// TwinCAT 3 PLC project SlaveController
// ProgramVersion: 3.1.4024.0
// libraries:
//   Tc2_EtherCAT, * (Beckhoff Automation GmbH)
//   Tc2_Math, * (Beckhoff Automation GmbH)
//   Tc2_Standard, * (Beckhoff Automation GmbH)
//   Tc2_System, * (Beckhoff Automation GmbH)
//   Tc2_Utilities, * (Beckhoff Automation GmbH)
//   Tc3_Module, * (Beckhoff Automation GmbH)
// project tree:
//   AgiMaths/Frames/ DHTrans.TcPOU, invFrame.TcPOU (not stored), rotX.TcPOU, rotY.TcPOU (not stored), rotZ.TcPOU (not stored), transform.TcPOU (not stored)
//   AgiMaths/MatrixLib/ angAxis2Rot.TcPOU, cross.TcPOU (not stored), Det5.TcPOU (not stored), Det6.TcPOU (not stored), Det7.TcPOU (not stored), invMat2.TcPOU, invMat6.TcPOU (not stored), invMat6Old.TcPOU (not stored), invMat3.TcPOU (not stored), invMat7.TcPOU, Mat3T.TcPOU (not stored), matAdd.TcPOU, matMultiNum.TcPOU (not stored), matMultiply.TcPOU (not stored), matMultiVec.TcPOU (not stored), matSelfAdd.TcPOU (not stored), vecDot.TcPOU (not stored), vecSelfAdd.TcPOU, matSelfSub.TcPOU (not stored), matSub.TcPOU (not stored), matTranspose.TcPOU (not stored), rot2AngAxis.TcPOU, vecAdd.TcPOU (not stored), norm.TcPOU, normalize.TcPOU, vecSelfMultiNum.TcPOU (not stored), vecMultiNum.TcPOU, vecSelfSub.TcPOU (not stored), vecSub.TcPOU (not stored)
//   AgiMaths/ sign.TcPOU (not stored), addVec7.TcPOU (not stored), atan2.TcPOU (not stored), cot.TcPOU (not stored)
//   DUTs/Enum/ E_ArmLightCtrlWord.TcDUT, E_CartJointState.TcDUT, E_EndoscopeType.TcDUT, E_EndoscopePosture.TcDUT, E_InstrumentType.TcDUT, E_MasterArmState.TcDUT, E_MatchedSlaveArmIdx.TcDUT (not stored), E_SetupArmState.TcDUT, E_SlaveArmState.TcDUT, E_DriverCtrlWord.TcDUT, E_DriverOPMode.TcDUT, E_DriverStatusWord.TcDUT
//   DUTs/Structure/MasterSlaveCommunication/ ST_MasterStatus.TcDUT, ST_SlaveStatus.TcDUT
//   DUTs/Structure/ ST_CartInputDataPool.TcDUT, ST_EtherCATState.TcDUT (not stored), ST_InstruOnChipData.TcDUT, ST_InstruStatus.TcDUT (not stored), ST_InstruTypeInfo.TcDUT, ST_SetupArmCtrlCmds.TcDUT (not stored), ST_SetupInputDataPool.TcDUT, ST_SlaveArmCtrlCmds.TcDUT, ST_SlaveInputDataPool.TcDUT, ST_Frame.TcDUT (not stored)
//   DUTs/Structure/TasksCommunication/ ST_CartJointData.TcDUT, ST_CartMotorInput.TcDUT, ST_CartMotorOutput.TcDUT, ST_CartStatus.TcDUT, ST_CartUIData.TcDUT, ST_SetupStatus.TcDUT, ST_SetupJointData.TcDUT, ST_SlaveDynaData.TcDUT, ST_SlaveUIData.TcDUT, ST_MasterJointData.TcDUT, ST_MotorInputs.TcDUT, ST_MotorOutputs.TcDUT, ST_SlaveJointData.TcDUT, ST_SafetyData.TcDUT
//   DUTs/Structure/UICommunication/ ST_cartOperation.TcDUT, ST_instruInfomation.TcDUT, ST_robotStateMachine.TcDUT, ST_uiControl.TcDUT
//   DUTs/Type/ Mat23.TcDUT, Mat2d.TcDUT, Mat32.TcDUT, Mat34.TcDUT (not stored), Mat53.TcDUT, Mat37.TcDUT (not stored), Mat43.TcDUT (not stored), Mat45.TcDUT (not stored), Mat35.TcDUT, Mat4d.TcDUT (not stored), Mat5d.TcDUT (not stored), Mat67.TcDUT (not stored), Mat6d.TcDUT (not stored), Mat76.TcDUT (not stored), Mat7d.TcDUT (not stored), Vec13d.TcDUT, Vec13di.TcDUT, Vec2d.TcDUT, Vec2i.TcDUT, Vec3i.TcDUT, Vec4b.TcDUT, Vec4d.TcDUT (not stored), Vec4i.TcDUT (not stored), Vec5b.TcDUT (not stored), Vec5d.TcDUT (not stored), Vec5i.TcDUT (not stored), Vec6b.TcDUT, Vec6i.TcDUT (not stored), Vec8b.TcDUT, Vec8d.TcDUT (not stored), Vec8di.TcDUT, Vec8i.TcDUT, Mat3d.TcDUT (not stored), Vec3d.TcDUT (not stored), Vec6d.TcDUT (not stored), Vec7d.TcDUT (not stored), Vec7i.TcDUT (not stored)
//   FBs_Auxiliary/ FB_cartJntDisenableDetect.TcPOU, FB_cartJntEnableDetect.TcPOU, FB_InstruNearDetect.TcPOU, FB_IOCheck.TcPOU, FB_IOToggleCheck.TcPOU, FB_rotaButtonDetect.TcPOU, FB_setupAdjustDetect.TcPOU, FB_setupJnt5AdjustDetect.TcPOU, FB_masterConnectionCheck.TcPOU, FB_TON.TcPOU (not stored), FB_trocarDetect.TcPOU, FB_PanelDetect.TcPOU (not stored), FB_InstrumentDetect.TcPOU, FB_AdjustDetect.TcPOU
//   FBs_BasicControllers/ FB_dither.TcPOU, FB_BasicInstruControl.TcPOU, FBMacroJntControl.TcPOU, FB_UltrosonicKnifeControl.TcPOU, FB_PID.TcPOU (not stored)
//   FBs_CartControlles/ FB_CartCtrlAdjust.TcPOU, FB_CartCtrlAsepticDeploy.TcPOU, FB_CartCtrlBase.TcPOU, FB_CartCtrlError.TcPOU, FB_CartCtrlInit.TcPOU, FB_CartCtrlInSurgery.TcPOU, FB_CartCtrlMotionCar.TcPOU, FB_CartCtrlReady.TcPOU, FB_CartCtrlRotaOverhang.TcPOU, FB_CartCtrlSlowDown.TcPOU, FB_CartCtrlStandColuAdjust.TcPOU, FB_CartPinDeploy.TcPOU, I_CartJointCtrl.TcIO
//   FBs_RobotDynamics/ FB_FullArmKinematic.TcPOU, FB_InstruViewCheck.TcPOU, FB_SlaveDynamic.TcPOU, FB_SlaveGravity.TcPOU, FB_SetupGravity.TcPOU
//   FBs_Robots/ FB_CartJoint.TcPOU, FB_CartRobot.TcPOU, FB_Instrument.TcPOU, FB_JointBase.TcPOU, FB_SetupArm.TcPOU, FB_SlaveCart.TcPOU, FB_SlaveJoint.TcPOU, FB_SetupJoint.TcPOU, FB_SetupRobot.TcPOU, FB_SlaveArm.TcPOU, FB_SlaveRobot.TcPOU
//   FBs_SetupControllers/ FB_SetupCtrlDisable.TcPOU, FB_SetupCtrlJnt5GraCali.TcPOU, FB_SetupCtrlHold.TcPOU, FB_SetupCtrlManualAdjust.TcPOU, FB_SetupCtrlPerformance.TcPOU, FB_SetupArmCtrlBase.TcPOU, FB_SetupCtrlAutoAdjust.TcPOU, FB_SetupCtrlCart.TcPOU (not stored), FB_SetupCtrlError.TcPOU, FB_SetupCtrlJnt3GraCali.TcPOU, FB_SetupCtrlInit.TcPOU, FB_SetupCtrlPackage.TcPOU (not stored), FB_SetupCtrlSelfCheck.TcPOU, I_SetupArmCtrl.TcIO (not stored)
//   FBs_SlaveControllers/ FB_SlaveCtrlDisable.TcPOU, FB_SlaveCtrlInstruInvasion.TcPOU, FB_SlaveCtrlInstruRetract.TcPOU, FB_SlaveCtrlInstruCali.TcPOU, FB_SlaveCtrlPerformance.TcPOU, FB_SlaveCtrlScopeToggle.TcPOU, FB_SlaveCtrlStop.TcPOU, FB_SlaveCtrlTest.TcPOU, FB_SlaveCtrlPackage.TcPOU, FB_SlaveCtrlEndoscope.TcPOU, FB_SlaveCtrlCart.TcPOU, FB_SlaveCtrlScopeReady.TcPOU, FB_SlaveCtrlSelfCheck.TcPOU, FB_SlaveCtrlError.TcPOU, FB_SlaveCtrlInstruReady.TcPOU, FB_SlaveCtrlMasterSlave.TcPOU, FB_SlaveCtrlMountInstru.TcPOU, FB_SlaveCtrlAdjust.TcPOU, FB_SlaveCtrlMountPanel.TcPOU, FB_SlaveCtrlPanelReady.TcPOU, FB_SlaveCtrlGraCali.TcPOU, FB_SlaveCtrlInit.TcPOU, FB_SlaveCtrlStandBy.TcPOU, FB_SlaveArmCtrlBase.TcPOU, I_SlaveArmCtrl.TcIO
//   FBs_TrajectoryPlanning/ FB_BasicDoubleS.TcPOU (not stored), FB_trajBase.TcPOU (not stored), FB_TrajMoveJ.TcPOU, FB_setupTrajMoveJ.TcPOU, linear_trajectory_with_quintic_polynomial_blends.TcPOU (not stored), quintic_spline_curve.TcPOU (not stored), Quintic_spline_curve_factor.TcPOU (not stored), TrapezoIDal_velocity_trajectory.TcPOU (not stored)
//   FBs_TrajectoryPlanning/OTG/ FB_secOrdTrajFilter.TcPOU (not stored), FB_thirdOrdTrajFilter.TcPOU (not stored)
//   FBs_Filters/ FB_LowPassFilter.TcPOU (not stored)
//   GVLs/CartJoints/ GVL_CartControlParameters.TcGVL, GVL_CartJointEncoderCaliData.TcGVL, GVL_CartMotorParameters.TcGVL
//   GVLs/configs/robot3/ GVL_CartJointEncoderCaliData_3.TcGVL, GVL_SetupArmDynamics_3.TcGVL, GVL_SlaveArmDynamics_3.TcGVL, GVL_SetupJointEncoderCaliData_3.TcGVL, GVL_SlaveJointEncoderCaliData_3.TcGVL
//   GVLs/configs/robot5/ GVL_CartJointEncoderCaliData_5.TcGVL, GVL_SetupArmDynamics_5.TcGVL, GVL_SlaveArmDynamics_5.TcGVL, GVL_SetupJointEncoderCaliData_5.TcGVL, GVL_SlaveJointEncoderCaliData_5.TcGVL
//   GVLs/configs/robot4/ GVL_SetupArmDynamics_4.TcGVL, GVL_SetupJointEncoderCaliData_4.TcGVL (not stored), GVL_SlaveArmDynamics_4.TcGVL, GVL_SlaveJointEncoderCaliData_4.TcGVL
//   GVLs/configs/robot6/ GVL_CartJointEncoderCaliData_6.TcGVL, GVL_SetupArmDynamics_6.TcGVL, GVL_SetupJointEncoderCaliData_6.TcGVL, GVL_SlaveArmDynamics_6.TcGVL, GVL_SlaveJointEncoderCaliData_6.TcGVL
//   GVLs/ GVL_interactUI.TcGVL, GVL_MathDefine.TcGVL, GVL_SafetyLogData.TcGVL, GVL_SafetyParameters.TcGVL, GVL_SystemParameters.TcGVL
//   GVLs/Instrument/ GVL_InstruCtrlParams.TcGVL, GVL_InstruTypeDefine.TcGVL
//   GVLs/SetupArms/ GVL_SetupArmDynamics.TcGVL, GVL_SetupJointEncoderCaliData.TcGVL, GVL_SetupMotorParameters.TcGVL, GVL_SetupArmKinematic.TcGVL, GVL_SetupControlParameters.TcGVL
//   GVLs/SlaveArms/ GVL_SlaveArmDynamics.TcGVL, GVL_SlaveArmKinematic.TcGVL, GVL_SlaveControlParameters.TcGVL, GVL_SlaveJointEncoderCaliData.TcGVL, GVL_SlaveMotorParameters.TcGVL
//   Mains/ CartControl.TcPOU, SafetyCheck.TcPOU, SetupArmControl.TcPOU (not stored), SlaveArmControl.TcPOU, RobotDynamics.TcPOU
//   SafetyCheck/ ASSERT.TcPOU, Fb_dataRecord.TcPOU, FB_EtherCATCheck.TcPOU (not stored), Fb_SafetyCheck.TcPOU, FB_Writer.TcPOU (not stored)
//   SafetyCheck/ErrRecord/ checkDelay.TcDUT, checkDelayTime.TcDUT, checkInputVariable.TcDUT, checkPermit.TcDUT, ST_Buffer.TcDUT, T_Buffer.TcDUT
//   Sandbox/ FB_SetupArmCheck.TcPOU (not stored), FB_SlaveArmCheck.TcPOU, FB_SlaveCtrlAdjust_bak1.TcPOU, FB_SlaveCtrlMasterSlave_bak1.TcPOU, FB_SlaveCtrlMasterSlave_bak2.TcPOU
//   Sandbox/knifeCmdPoseTest/ atan2_function.TcPOU, FB_CSVWrite.TcPOU, knifePoseSelect.TcPOU, tr_to_rpy.TcPOU, tr_to_space_vector.TcPOU
//   / TaskCartControl.TcTTO, TaskDynamic.TcTTO (not stored), TaskSafetyCheck.TcTTO, TaskSetupArmControl.TcTTO (not stored), TaskSlaveArmControl.TcTTO
// real-time tasks:
//   TASK TaskSlaveArmControl: cycle T#250us, priority 1, ADS port 350
//   TASK TaskDynamic: cycle T#1ms, priority 2, ADS port 351
//   TASK TaskSetupArmControl: cycle T#1ms, priority 3, ADS port 352
//   TASK TaskSafetyCheck: cycle T#1ms, priority 6, ADS port 353
//   TASK TaskCartControl: cycle T#1ms, priority 4, ADS port 354
// I/O:
//   DEVICE Device 5 (RT-Ethernet Adapter)
//   DEVICE MSCommunication, AmsNetId 169.254.186.39.2.1
//     Term 20 (EK1100) [EK1100 EtherCAT Coupler (2A E-Bus)]
//       Term 21 (EL6695) [EL6695 EtherCAT Bridge terminal (Primary)]
//       Term 8 (EL9011) [EL9011 End Terminal]
//     Term 22 (EK1100) [EK1100 EtherCAT Coupler (2A E-Bus)]
//       Term 23 (EL6070) [EL6070 1Ch. Licensing-Terminal]
//       Term 24 (EL1008) [EL1008 8Ch. Dig. Input 24V, 3ms]
//       Term 25 (EL2008) [EL2008 8Ch. Dig. Output 24V, 0.5A]
//       Term 26 (EL3004) [EL3004 4Ch. Ana. Input +/-10V]
//       Term 9 (EL9011) [EL9011 End Terminal]
//   DEVICE SlaveArm1, AmsNetId 169.254.186.39.3.1
//     Box 29 (CU2508) [CU2508 Ethernet Port]
//     SetupJoint12 [AX58200_MotorControl]
//     SetupJoint3 [AX58200_MotorControl]
//     SetupJoint4 [AX58200_MotorControl]
//     SetupJoint5 [AX58200_MotorControl]
//     SlaveJoint1 [AX58200_MotorControl]
//     SlaveJoint2 [AX58200_MotorControl]
//     SlaveJoint3 [AX58200_MotorControl]
//     SlaveJoint45 [AX58200_MotorControl]
//     SlaveJoint678 [AX58200_MotorControl]
//   DEVICE SlaveArm2, AmsNetId 169.254.186.39.8.1
//     Box 39 (CU2508) [CU2508 Ethernet Port]
//     SetupJoint12 [AX58200_MotorControl]
//     SetupJoint3 [AX58200_MotorControl]
//     SetupJoint4 [AX58200_MotorControl]
//     SetupJoint5 [AX58200_MotorControl]
//     SlaveJoint1 [AX58200_MotorControl]
//     SlaveJoint2 [AX58200_MotorControl]
//     SlaveJoint3 [AX58200_MotorControl]
//     SlaveJoint45 [AX58200_MotorControl]
//     SlaveJoint678 [AX58200_MotorControl]
//   DEVICE SlaveArm3, AmsNetId 169.254.186.39.9.1
//     Box 49 (CU2508) [CU2508 Ethernet Port]
//     SetupJoint12 [AX58200_MotorControl]
//     SetupJoint3 [AX58200_MotorControl]
//     SetupJoint4 [AX58200_MotorControl]
//     SetupJoint5 [AX58200_MotorControl]
//     SlaveJoint1 [AX58200_MotorControl]
//     SlaveJoint2 [AX58200_MotorControl]
//     SlaveJoint3 [AX58200_MotorControl]
//     SlaveJoint45 [AX58200_MotorControl]
//     SlaveJoint678 [AX58200_MotorControl]
//   DEVICE SlaveArm4, AmsNetId 169.254.186.39.10.1
//     Box 59 (CU2508) [CU2508 Ethernet Port]
//     SetupJoint12 [AX58200_MotorControl]
//     SetupJoint3 [AX58200_MotorControl]
//     SetupJoint4 [AX58200_MotorControl]
//     SetupJoint5 [AX58200_MotorControl]
//     SlaveJoint1 [AX58200_MotorControl]
//     SlaveJoint2 [AX58200_MotorControl]
//     SlaveJoint3 [AX58200_MotorControl_3AxiS]
//     SlaveJoint45 [AX58200_MotorControl_3AxiS]
//     SlaveJoint678 [AX58200_MotorControl_3AxiS]
//   DEVICE Cart, AmsNetId 169.254.186.39.4.1
//     CartJnt5 [iPOS8015 BZ-CAT]
//     CartJnt3 [iPOS4850 BX-CAT]
//     CartJnt4 [iPOS4850 BX-CAT]
//     CartJnt1 [AX58200_MotorControl]
//     CartJnt2 [AX58200_MotorControl]
//     CartJnt6 [AX58200_MotorControl]
//     CartJnt7 [AX58200_MotorControl]
//     CartJnt8 [AX58200_MotorControl]
// variable links:
//   SlaveController/SlaveController Instance <-> Cart/CartJnt1
//     TaskCartControl Inputs/CartControl.m_cartRobot.m_slaveCart.m_cartJoints[1].m_motorInputs/m_current <-> TxPdoMappingCspCsv/Torque actual value
//     TaskCartControl Inputs/CartControl.m_cartRobot.m_slaveCart.m_cartJoints[1].m_motorInputs/m_driverError <-> TxPdoMappingCspCsv/digital input
//     TaskCartControl Inputs/CartControl.m_cartRobot.m_slaveCart.m_cartJoints[1].m_motorInputs/m_motorEncoder <-> TxPdoMappingCspCsv/Position actual value
//     TaskCartControl Inputs/CartControl.m_cartRobot.m_slaveCart.m_cartJoints[1].m_motorInputs/m_statusWord <-> TxPdoMappingCspCsv/Statusword
//     TaskCartControl Outputs/CartControl.m_cartRobot.m_slaveCart.m_cartJoints[1].m_motorOutputs/m_cmdCurrent <-> RxPdoMappingCspCsv/Target torque
//     TaskCartControl Outputs/CartControl.m_cartRobot.m_slaveCart.m_cartJoints[1].m_motorOutputs/m_cmdMotorEncoder <-> RxPdoMappingCspCsv/Target position
//     TaskCartControl Outputs/CartControl.m_cartRobot.m_slaveCart.m_cartJoints[1].m_motorOutputs/m_controlWord <-> RxPdoMappingCspCsv/Controlword
//     TaskCartControl Outputs/CartControl.m_cartRobot.m_slaveCart.m_cartJoints[1].m_motorOutputs/m_opMode <-> RxPdoMappingCspCsv/Modes of operation
//   SlaveController/SlaveController Instance <-> Cart/CartJnt2
//     TaskCartControl Inputs/CartControl.m_cartRobot.m_slaveCart.m_cartJoints[2].m_motorInputs/m_current <-> TxPdoMappingCspCsv/Torque actual value
//     TaskCartControl Inputs/CartControl.m_cartRobot.m_slaveCart.m_cartJoints[2].m_motorInputs/m_driverError <-> TxPdoMappingCspCsv/digital input
//     TaskCartControl Inputs/CartControl.m_cartRobot.m_slaveCart.m_cartJoints[2].m_motorInputs/m_motorEncoder <-> TxPdoMappingCspCsv/Position actual value
//     TaskCartControl Inputs/CartControl.m_cartRobot.m_slaveCart.m_cartJoints[2].m_motorInputs/m_statusWord <-> TxPdoMappingCspCsv/Statusword
//     TaskCartControl Inputs/CartControl.m_cartRobot.m_slaveCart.m_cartJoints[5].m_motorInputs/m_linkEncoder <-> TxPdoMappingCspCsv/ENC2
//     TaskCartControl Outputs/CartControl.m_cartRobot.m_slaveCart.m_cartJoints[2].m_motorOutputs/m_cmdCurrent <-> RxPdoMappingCspCsv/Target torque
//     TaskCartControl Outputs/CartControl.m_cartRobot.m_slaveCart.m_cartJoints[2].m_motorOutputs/m_cmdMotorEncoder <-> RxPdoMappingCspCsv/Target position
//     TaskCartControl Outputs/CartControl.m_cartRobot.m_slaveCart.m_cartJoints[2].m_motorOutputs/m_controlWord <-> RxPdoMappingCspCsv/Controlword
//     TaskCartControl Outputs/CartControl.m_cartRobot.m_slaveCart.m_cartJoints[2].m_motorOutputs/m_opMode <-> RxPdoMappingCspCsv/Modes of operation
//   SlaveController/SlaveController Instance <-> Cart/CartJnt3
//     TaskCartControl Inputs/CartControl.m_cartRobot.m_slaveCart.m_cartJoints[3].m_motorInputs/m_motorEncoder <-> Transmit PDO 1 mapping parameters/Position actual value
//     TaskCartControl Inputs/CartControl.m_cartRobot.m_slaveCart.m_cartJoints[3].m_motorInputs/m_statusWord <-> Transmit PDO 1 mapping parameters/Statusword
//     TaskCartControl Outputs/CartControl.m_cartRobot.m_slaveCart.m_cartJoints[3].m_cartMotorOutput/m_cmdAccMz <-> Receive PDO 4 mapping parameters/Profile acceleration
//     TaskCartControl Outputs/CartControl.m_cartRobot.m_slaveCart.m_cartJoints[3].m_cartMotorOutput/m_cmdVelMz <-> Receive PDO 4 mapping parameters/Profile velocity
//     TaskCartControl Outputs/CartControl.m_cartRobot.m_slaveCart.m_cartJoints[3].m_cartMotorOutput/m_cmdVelMzVelMode <-> Receive PDO 3 mapping parameters/Target Velocity
//     TaskCartControl Outputs/CartControl.m_cartRobot.m_slaveCart.m_cartJoints[3].m_motorOutputs/m_cmdMotorEncoder <-> Receive PDO 1 mapping parameters/Target position
//     TaskCartControl Outputs/CartControl.m_cartRobot.m_slaveCart.m_cartJoints[3].m_motorOutputs/m_controlWord <-> Receive PDO 1 mapping parameters/Controlword
//     TaskCartControl Outputs/CartControl.m_cartRobot.m_slaveCart.m_cartJoints[3].m_motorOutputs/m_opMode <-> Receive PDO 3 mapping parameters/Modes of operation
//   SlaveController/SlaveController Instance <-> Cart/CartJnt4
//     TaskCartControl Inputs/CartControl.m_cartRobot.m_slaveCart.m_cartJoints[4].m_motorInputs/m_motorEncoder <-> Transmit PDO 1 mapping parameters/Position actual value
//     TaskCartControl Inputs/CartControl.m_cartRobot.m_slaveCart.m_cartJoints[4].m_motorInputs/m_statusWord <-> Transmit PDO 1 mapping parameters/Statusword
//     TaskCartControl Outputs/CartControl.m_cartRobot.m_slaveCart.m_cartJoints[4].m_cartMotorOutput/m_cmdAccMz <-> Receive PDO 4 mapping parameters/Profile acceleration
//     TaskCartControl Outputs/CartControl.m_cartRobot.m_slaveCart.m_cartJoints[4].m_cartMotorOutput/m_cmdVelMz <-> Receive PDO 4 mapping parameters/Profile velocity
//     TaskCartControl Outputs/CartControl.m_cartRobot.m_slaveCart.m_cartJoints[4].m_cartMotorOutput/m_cmdVelMzVelMode <-> Receive PDO 3 mapping parameters/Target  Velocity
//     TaskCartControl Outputs/CartControl.m_cartRobot.m_slaveCart.m_cartJoints[4].m_motorOutputs/m_cmdMotorEncoder <-> Receive PDO 1 mapping parameters/Target position
//     TaskCartControl Outputs/CartControl.m_cartRobot.m_slaveCart.m_cartJoints[4].m_motorOutputs/m_controlWord <-> Receive PDO 1 mapping parameters/Controlword
//     TaskCartControl Outputs/CartControl.m_cartRobot.m_slaveCart.m_cartJoints[4].m_motorOutputs/m_opMode <-> Receive PDO 3 mapping parameters/Modes of operation
//   SlaveController/SlaveController Instance <-> Cart/CartJnt5
//     TaskCartControl Inputs/CartControl.m_cartRobot.m_slaveCart.m_cartJoints[5].m_motorInputs/m_motorEncoder <-> Transmit PDO 1 mapping parameters/Position actual value
//     TaskCartControl Inputs/CartControl.m_cartRobot.m_slaveCart.m_cartJoints[5].m_motorInputs/m_statusWord <-> Transmit PDO 1 mapping parameters/Statusword
//     TaskCartControl Outputs/CartControl.m_cartRobot.m_slaveCart.m_cartJoints[5].m_cartMotorOutput/m_cmdAccMz <-> Receive PDO 4 mapping parameters/Profile acceleration
//     TaskCartControl Outputs/CartControl.m_cartRobot.m_slaveCart.m_cartJoints[5].m_cartMotorOutput/m_cmdVelMz <-> Receive PDO 4 mapping parameters/Profile velocity
//     TaskCartControl Outputs/CartControl.m_cartRobot.m_slaveCart.m_cartJoints[5].m_cartMotorOutput/m_cmdVelMzVelMode <-> Receive PDO 3 mapping parameters/Target Velocity
//     TaskCartControl Outputs/CartControl.m_cartRobot.m_slaveCart.m_cartJoints[5].m_motorOutputs/m_cmdMotorEncoder <-> Receive PDO 1 mapping parameters/Target position
//     TaskCartControl Outputs/CartControl.m_cartRobot.m_slaveCart.m_cartJoints[5].m_motorOutputs/m_controlWord <-> Receive PDO 1 mapping parameters/Controlword
//     TaskCartControl Outputs/CartControl.m_cartRobot.m_slaveCart.m_cartJoints[5].m_motorOutputs/m_opMode <-> Receive PDO 3 mapping parameters/Modes of operation
//   SlaveController/SlaveController Instance <-> Cart/CartJnt6
//     TaskCartControl Inputs/CartControl.m_cartRobot.m_slaveCart.m_cartJoints[6].m_motorInputs/m_current <-> TxPdoMappingCspCsv/Torque actual value
//     TaskCartControl Inputs/CartControl.m_cartRobot.m_slaveCart.m_cartJoints[6].m_motorInputs/m_driverError <-> TxPdoMappingCspCsv/digital input
//     TaskCartControl Inputs/CartControl.m_cartRobot.m_slaveCart.m_cartJoints[6].m_motorInputs/m_linkEncoder <-> TxPdoMappingCspCsv/ENC2
//     TaskCartControl Inputs/CartControl.m_cartRobot.m_slaveCart.m_cartJoints[6].m_motorInputs/m_motorEncoder <-> TxPdoMappingCspCsv/Position actual value
//     TaskCartControl Inputs/CartControl.m_cartRobot.m_slaveCart.m_cartJoints[6].m_motorInputs/m_statusWord <-> TxPdoMappingCspCsv/Statusword
//     TaskCartControl Outputs/CartControl.m_cartRobot.m_openHorizonLaser <-> RxPdoMappingCspCsv/Target velocity
//     TaskCartControl Outputs/CartControl.m_cartRobot.m_slaveCart.m_cartJoints[6].m_motorOutputs/m_cmdCurrent <-> RxPdoMappingCspCsv/Target torque
//     TaskCartControl Outputs/CartControl.m_cartRobot.m_slaveCart.m_cartJoints[6].m_motorOutputs/m_cmdMotorEncoder <-> RxPdoMappingCspCsv/Target position
//     TaskCartControl Outputs/CartControl.m_cartRobot.m_slaveCart.m_cartJoints[6].m_motorOutputs/m_controlWord <-> RxPdoMappingCspCsv/Controlword
//     TaskCartControl Outputs/CartControl.m_cartRobot.m_slaveCart.m_cartJoints[6].m_motorOutputs/m_opMode <-> RxPdoMappingCspCsv/Modes of operation
//   SlaveController/SlaveController Instance <-> Cart/CartJnt7
//     TaskCartControl Inputs/CartControl.m_cartRobot.m_slaveCart.m_cartJoints[7].m_motorInputs/m_current <-> TxPdoMappingCspCsv/Torque actual value
//     TaskCartControl Inputs/CartControl.m_cartRobot.m_slaveCart.m_cartJoints[7].m_motorInputs/m_driverError <-> TxPdoMappingCspCsv/digital input
//     TaskCartControl Inputs/CartControl.m_cartRobot.m_slaveCart.m_cartJoints[7].m_motorInputs/m_linkEncoder <-> TxPdoMappingCspCsv/ENC2
//     TaskCartControl Inputs/CartControl.m_cartRobot.m_slaveCart.m_cartJoints[7].m_motorInputs/m_motorEncoder <-> TxPdoMappingCspCsv/Position actual value
//     TaskCartControl Inputs/CartControl.m_cartRobot.m_slaveCart.m_cartJoints[7].m_motorInputs/m_statusWord <-> TxPdoMappingCspCsv/Statusword
//     TaskCartControl Outputs/CartControl.m_cartRobot.m_slaveCart.m_cartJoints[7].m_motorOutputs/m_cmdCurrent <-> RxPdoMappingCspCsv/Target torque
//     TaskCartControl Outputs/CartControl.m_cartRobot.m_slaveCart.m_cartJoints[7].m_motorOutputs/m_cmdMotorEncoder <-> RxPdoMappingCspCsv/Target position
//     TaskCartControl Outputs/CartControl.m_cartRobot.m_slaveCart.m_cartJoints[7].m_motorOutputs/m_controlWord <-> RxPdoMappingCspCsv/Controlword
//     TaskCartControl Outputs/CartControl.m_cartRobot.m_slaveCart.m_cartJoints[7].m_motorOutputs/m_opMode <-> RxPdoMappingCspCsv/Modes of operation
//   SlaveController/SlaveController Instance <-> Cart/CartJnt8
//     TaskCartControl Inputs/CartControl.m_cartRobot.m_slaveCart.m_cartJoints[8].m_motorInputs/m_current <-> TxPdoMappingCspCsv/Torque actual value
//     TaskCartControl Inputs/CartControl.m_cartRobot.m_slaveCart.m_cartJoints[8].m_motorInputs/m_driverError <-> TxPdoMappingCspCsv/digital input
//     TaskCartControl Inputs/CartControl.m_cartRobot.m_slaveCart.m_cartJoints[8].m_motorInputs/m_linkEncoder <-> TxPdoMappingCspCsv/ENC2
//     TaskCartControl Inputs/CartControl.m_cartRobot.m_slaveCart.m_cartJoints[8].m_motorInputs/m_motorEncoder <-> TxPdoMappingCspCsv/Position actual value
//     TaskCartControl Inputs/CartControl.m_cartRobot.m_slaveCart.m_cartJoints[8].m_motorInputs/m_statusWord <-> TxPdoMappingCspCsv/Statusword
//     TaskCartControl Outputs/CartControl.m_cartRobot.m_openCrossLaser <-> RxPdoMappingCspCsv/Target velocity
//     TaskCartControl Outputs/CartControl.m_cartRobot.m_slaveCart.m_cartJoints[8].m_motorOutputs/m_cmdCurrent <-> RxPdoMappingCspCsv/Target torque
//     TaskCartControl Outputs/CartControl.m_cartRobot.m_slaveCart.m_cartJoints[8].m_motorOutputs/m_cmdMotorEncoder <-> RxPdoMappingCspCsv/Target position
//     TaskCartControl Outputs/CartControl.m_cartRobot.m_slaveCart.m_cartJoints[8].m_motorOutputs/m_controlWord <-> RxPdoMappingCspCsv/Controlword
//     TaskCartControl Outputs/CartControl.m_cartRobot.m_slaveCart.m_cartJoints[8].m_motorOutputs/m_opMode <-> RxPdoMappingCspCsv/Modes of operation
//   SlaveController/SlaveController Instance <-> MSCommunication/Term 20 (EK1100)/Term 21 (EL6695)
//     TaskSafetyCheck Inputs/SafetyCheck.m_masterRobotData <-> IO Inputs/MasterRobotData
//     TaskSlaveArmControl Inputs/SlaveArmControl.m_masterRobotData <-> IO Inputs/MasterRobotData
//     TaskSlaveArmControl Outputs/SlaveArmControl.m_slaveRobotData <-> IO Outputs/SlaveRobotData
//   SlaveController/SlaveController Instance <-> MSCommunication/Term 22 (EK1100)/Term 24 (EL1008)
//     TaskCartControl Inputs/CartControl.m_cartRobot.m_carHandChassisDriveUnlock[1] <-> Channel 5/Input
//     TaskCartControl Inputs/CartControl.m_cartRobot.m_carHandChassisDriveUnlock[2] <-> Channel 6/Input
//     TaskCartControl Inputs/CartControl.m_cartRobot.m_slaveCart.m_drivingLeverSensorAuto <-> Channel 8/Input
//     TaskCartControl Inputs/CartControl.m_cartRobot.m_slaveCart.m_drivingLeverSensorManual <-> Channel 7/Input
//     TaskCartControl Inputs/CartControl.m_cartRobot.m_slaveCart.m_stabilizFootSensorLeft <-> Channel 3/Input
//     TaskCartControl Inputs/CartControl.m_cartRobot.m_slaveCart.m_stabilizFootSensorRight <-> Channel 4/Input
//     TaskSafetyCheck Inputs/SafetyCheck.m_emergencyStopButton <-> Channel 2/Input
//     TaskSlaveArmControl Inputs/SafetyCheck.m_stopButton <-> Channel 1/Input
//   SlaveController/SlaveController Instance <-> MSCommunication/Term 22 (EK1100)/Term 25 (EL2008)
//     TaskCartControl Outputs/CartControl.m_cartRobot.m_slaveCart.m_screwBreak <-> Channel 5/Output
//     TaskSafetyCheck Outputs/SafetyCheck.m_warningTone[{1..4}] <-> Channel {1..4}/Output  (4 links)
//   SlaveController/SlaveController Instance <-> MSCommunication/Term 22 (EK1100)/Term 26 (EL3004)
//     TaskCartControl Inputs/CartControl.m_cartRobot.m_slaveCart.m_driveForce[1] <-> AI Standard Channel 2/Value
//     TaskCartControl Inputs/CartControl.m_cartRobot.m_slaveCart.m_driveForce[2] <-> AI Standard Channel 1/Value
//   SlaveController/SlaveController Instance <-> SlaveArm1/SetupJoint12
//     TaskSetupArmControl Inputs/SetupArmControl.m_setupRobot.m_setupArms[1].m_joints[1].m_motorInputs/m_linkEncoder <-> TxPdoMappingCspCsv/ENC2
//     TaskSetupArmControl Inputs/SetupArmControl.m_setupRobot.m_setupArms[1].m_joints[1].m_motorInputs/m_statusWord <-> TxPdoMappingCspCsv/Statusword
//     TaskSetupArmControl Inputs/SetupArmControl.m_setupRobot.m_setupArms[1].m_joints[2].m_motorInputs/m_statusWord <-> TxPdoMappingCspCsv/Statusword
//     TaskSetupArmControl Inputs/SetupArmControl.m_setupRobot.m_setupArms[1].m_joints[2].m_motorInputs/m_linkEncoder <-> TxPdoMappingCspCsv/Torque actual value
//     TaskSetupArmControl Outputs/SetupArmControl.m_setupRobot.m_setupArms[1].m_joints[1].m_motorOutputs/m_controlWord <-> RxPdoMappingCspCsv/Controlword
//   SlaveController/SlaveController Instance <-> SlaveArm1/SetupJoint3
//     TaskSetupArmControl Inputs/SetupArmControl.m_setupRobot.m_setupArms[1].m_joints[3].m_motorInputs/m_current <-> TxPdoMappingCspCsv/Torque actual value
//     TaskSetupArmControl Inputs/SetupArmControl.m_setupRobot.m_setupArms[1].m_joints[3].m_motorInputs/m_linkEncoder <-> TxPdoMappingCspCsv/ENC2
//     TaskSetupArmControl Inputs/SetupArmControl.m_setupRobot.m_setupArms[1].m_joints[3].m_motorInputs/m_motorEncoder <-> TxPdoMappingCspCsv/Position actual value
//     TaskSetupArmControl Inputs/SetupArmControl.m_setupRobot.m_setupArms[1].m_joints[3].m_motorInputs/m_statusWord <-> TxPdoMappingCspCsv/Statusword
//     TaskSetupArmControl Outputs/SetupArmControl.m_setupRobot.m_setupArms[1].m_joints[3].m_motorOutputs/m_cmdCurrent <-> RxPdoMappingCspCsv/Target torque
//     TaskSetupArmControl Outputs/SetupArmControl.m_setupRobot.m_setupArms[1].m_joints[3].m_motorOutputs/m_cmdMotorEncoder <-> RxPdoMappingCspCsv/Target position
//     TaskSetupArmControl Outputs/SetupArmControl.m_setupRobot.m_setupArms[1].m_joints[3].m_motorOutputs/m_controlWord <-> RxPdoMappingCspCsv/Controlword
//     TaskSetupArmControl Outputs/SetupArmControl.m_setupRobot.m_setupArms[1].m_joints[3].m_motorOutputs/m_opMode <-> RxPdoMappingCspCsv/Modes of operation
//   SlaveController/SlaveController Instance <-> SlaveArm1/SetupJoint4
//     TaskSetupArmControl Inputs/SetupArmControl.m_setupRobot.m_setupArms[1].m_joints[4].m_motorInputs/m_current <-> TxPdoMappingCspCsv/Torque actual value
//     TaskSetupArmControl Inputs/SetupArmControl.m_setupRobot.m_setupArms[1].m_joints[4].m_motorInputs/m_motorEncoder <-> TxPdoMappingCspCsv/Position actual value
//     TaskSetupArmControl Inputs/SetupArmControl.m_setupRobot.m_setupArms[1].m_joints[4].m_motorInputs/m_statusWord <-> TxPdoMappingCspCsv/Statusword
//     TaskSetupArmControl Outputs/SetupArmControl.m_setupRobot.m_setupArms[1].m_joints[4].m_motorOutputs/m_cmdCurrent <-> RxPdoMappingCspCsv/Target torque
//     TaskSetupArmControl Outputs/SetupArmControl.m_setupRobot.m_setupArms[1].m_joints[4].m_motorOutputs/m_cmdMotorEncoder <-> RxPdoMappingCspCsv/Target position
//     TaskSetupArmControl Outputs/SetupArmControl.m_setupRobot.m_setupArms[1].m_joints[4].m_motorOutputs/m_controlWord <-> RxPdoMappingCspCsv/Controlword
//     TaskSetupArmControl Outputs/SetupArmControl.m_setupRobot.m_setupArms[1].m_joints[4].m_motorOutputs/m_opMode <-> RxPdoMappingCspCsv/Modes of operation
//   SlaveController/SlaveController Instance <-> SlaveArm1/SetupJoint5
//     TaskSetupArmControl Inputs/SetupArmControl.m_setupRobot.m_setupArms[1].m_joints[4].m_motorInputs/m_linkEncoder <-> TxPdoMappingCspCsv/ENC2
//     TaskSetupArmControl Inputs/SetupArmControl.m_setupRobot.m_setupArms[1].m_joints[5].m_motorInputs/m_current <-> TxPdoMappingCspCsv/Torque actual value
//     TaskSetupArmControl Inputs/SetupArmControl.m_setupRobot.m_setupArms[1].m_joints[5].m_motorInputs/m_linkEncoder <-> TxPdoMappingCspCsv/analog input
//     TaskSetupArmControl Inputs/SetupArmControl.m_setupRobot.m_setupArms[1].m_joints[5].m_motorInputs/m_motorEncoder <-> TxPdoMappingCspCsv/Position actual value
//     TaskSetupArmControl Inputs/SetupArmControl.m_setupRobot.m_setupArms[1].m_joints[5].m_motorInputs/m_statusWord <-> TxPdoMappingCspCsv/Statusword
//     TaskSetupArmControl Outputs/SetupArmControl.m_setupRobot.m_setupArms[1].m_joints[5].m_motorOutputs/m_cmdCurrent <-> RxPdoMappingCspCsv/Target torque
//     TaskSetupArmControl Outputs/SetupArmControl.m_setupRobot.m_setupArms[1].m_joints[5].m_motorOutputs/m_cmdMotorEncoder <-> RxPdoMappingCspCsv/Target position
//     TaskSetupArmControl Outputs/SetupArmControl.m_setupRobot.m_setupArms[1].m_joints[5].m_motorOutputs/m_controlWord <-> RxPdoMappingCspCsv/Controlword
//     TaskSetupArmControl Outputs/SetupArmControl.m_setupRobot.m_setupArms[1].m_joints[5].m_motorOutputs/m_opMode <-> RxPdoMappingCspCsv/Modes of operation
//   SlaveController/SlaveController Instance <-> SlaveArm1/SlaveJoint1
//     TaskSlaveArmControl Inputs/SlaveArmControl.m_slaveRobot.m_slaveArms[1].m_joints[1].m_motorInputs/m_current <-> TxPdoMappingCspCsv/Torque actual value
//     TaskSlaveArmControl Inputs/SlaveArmControl.m_slaveRobot.m_slaveArms[1].m_joints[1].m_motorInputs/m_linkEncoder <-> TxPdoMappingCspCsv/ENC2
//     TaskSlaveArmControl Inputs/SlaveArmControl.m_slaveRobot.m_slaveArms[1].m_joints[1].m_motorInputs/m_motorEncoder <-> TxPdoMappingCspCsv/Position actual value
//     TaskSlaveArmControl Inputs/SlaveArmControl.m_slaveRobot.m_slaveArms[1].m_joints[1].m_motorInputs/m_statusWord <-> TxPdoMappingCspCsv/Statusword
//     TaskSlaveArmControl Outputs/SlaveArmControl.m_slaveRobot.m_slaveArms[1].m_joints[1].m_motorOutputs/m_cmdCurrent <-> RxPdoMappingCspCsv/Target torque
//     TaskSlaveArmControl Outputs/SlaveArmControl.m_slaveRobot.m_slaveArms[1].m_joints[1].m_motorOutputs/m_cmdMotorEncoder <-> RxPdoMappingCspCsv/Target position
//     TaskSlaveArmControl Outputs/SlaveArmControl.m_slaveRobot.m_slaveArms[1].m_joints[1].m_motorOutputs/m_controlWord <-> RxPdoMappingCspCsv/Controlword
//     TaskSlaveArmControl Outputs/SlaveArmControl.m_slaveRobot.m_slaveArms[1].m_joints[1].m_motorOutputs/m_opMode <-> RxPdoMappingCspCsv/Modes of operation
//   SlaveController/SlaveController Instance <-> SlaveArm1/SlaveJoint2
//     TaskCartControl Inputs/CartControl.m_cartRobot.m_slaveCart.m_carRotaOverhangIO[1] <-> TxPdoMappingCspCsv/digital input
//     TaskSetupArmControl Outputs/SetupArmControl.m_setupRobot.m_setupArms[1].m_lightIO <-> RxPdoMappingCspCsv/Target velocity
//     TaskSlaveArmControl Inputs/SlaveArmControl.m_slaveRobot.m_slaveArms[1].m_joints[2].m_motorInputs/m_current <-> TxPdoMappingCspCsv/Torque actual value
//     TaskSlaveArmControl Inputs/SlaveArmControl.m_slaveRobot.m_slaveArms[1].m_joints[2].m_motorInputs/m_linkEncoder <-> TxPdoMappingCspCsv/ENC2
//     TaskSlaveArmControl Inputs/SlaveArmControl.m_slaveRobot.m_slaveArms[1].m_joints[2].m_motorInputs/m_motorEncoder <-> TxPdoMappingCspCsv/Position actual value
//     TaskSlaveArmControl Inputs/SlaveArmControl.m_slaveRobot.m_slaveArms[1].m_joints[2].m_motorInputs/m_statusWord <-> TxPdoMappingCspCsv/Statusword
//     TaskSlaveArmControl Outputs/SlaveArmControl.m_slaveRobot.m_slaveArms[1].m_joints[2].m_motorOutputs/m_cmdCurrent <-> RxPdoMappingCspCsv/Target torque
//     TaskSlaveArmControl Outputs/SlaveArmControl.m_slaveRobot.m_slaveArms[1].m_joints[2].m_motorOutputs/m_cmdMotorEncoder <-> RxPdoMappingCspCsv/Target position
//     TaskSlaveArmControl Outputs/SlaveArmControl.m_slaveRobot.m_slaveArms[1].m_joints[2].m_motorOutputs/m_controlWord <-> RxPdoMappingCspCsv/Controlword
//     TaskSlaveArmControl Outputs/SlaveArmControl.m_slaveRobot.m_slaveArms[1].m_joints[2].m_motorOutputs/m_opMode <-> RxPdoMappingCspCsv/Modes of operation
//   SlaveController/SlaveController Instance <-> SlaveArm1/SlaveJoint3
//     TaskCartControl Inputs/CartControl.m_cartRobot.m_slaveCart.m_trocarIO[1] <-> TxPdoMappingCspCsv/digital input
//     TaskSetupArmControl Inputs/SetupArmControl.m_setupRobot.m_setupArms[1].m_adjustIO <-> TxPdoMappingCspCsv/digital input
//     TaskSlaveArmControl Inputs/SlaveArmControl.m_slaveRobot.m_slaveArms[1].m_adjustIO <-> TxPdoMappingCspCsv/digital input
//     TaskSlaveArmControl Inputs/SlaveArmControl.m_slaveRobot.m_slaveArms[1].m_joints[3].m_motorInputs/m_current <-> TxPdoMappingCspCsv/Torque actual value
//     TaskSlaveArmControl Inputs/SlaveArmControl.m_slaveRobot.m_slaveArms[1].m_joints[3].m_motorInputs/m_linkEncoder <-> TxPdoMappingCspCsv/ENC2 for aix1
//     TaskSlaveArmControl Inputs/SlaveArmControl.m_slaveRobot.m_slaveArms[1].m_joints[3].m_motorInputs/m_motorEncoder <-> TxPdoMappingCspCsv/Position actual value
//     TaskSlaveArmControl Inputs/SlaveArmControl.m_slaveRobot.m_slaveArms[1].m_joints[3].m_motorInputs/m_statusWord <-> TxPdoMappingCspCsv/Statusword
//     TaskSlaveArmControl Outputs/SlaveArmControl.m_slaveRobot.m_slaveArms[1].m_joints[3].m_motorOutputs/m_cmdCurrent <-> RxPdoMappingCspCsv/Target Torque value
//     TaskSlaveArmControl Outputs/SlaveArmControl.m_slaveRobot.m_slaveArms[1].m_joints[3].m_motorOutputs/m_cmdMotorEncoder <-> RxPdoMappingCspCsv/Target position
//     TaskSlaveArmControl Outputs/SlaveArmControl.m_slaveRobot.m_slaveArms[1].m_joints[3].m_motorOutputs/m_controlWord <-> RxPdoMappingCspCsv/Controlword
//     TaskSlaveArmControl Outputs/SlaveArmControl.m_slaveRobot.m_slaveArms[1].m_joints[3].m_motorOutputs/m_opMode <-> RxPdoMappingCspCsv/Modes of operation
//   SlaveController/SlaveController Instance <-> SlaveArm1/SlaveJoint45
//     TaskSlaveArmControl Inputs/SlaveArmControl.m_slaveRobot.m_slaveArms[1].m_joints[4].m_motorInputs/m_current <-> TxPdoMappingCspCsv/Velocity actual value for aix2
//     TaskSlaveArmControl Inputs/SlaveArmControl.m_slaveRobot.m_slaveArms[1].m_joints[4].m_motorInputs/m_linkEncoder <-> TxPdoMappingCspCsv/ENC2 for aix2
//     TaskSlaveArmControl Inputs/SlaveArmControl.m_slaveRobot.m_slaveArms[1].m_joints[5].m_motorInputs/m_linkEncoder <-> TxPdoMappingCspCsv/ENC2 for aix3
//     TaskSlaveArmControl Inputs/SlaveArmControl.m_slaveRobot.m_slaveArms[1].m_joints[4].m_motorInputs/m_motorEncoder <-> TxPdoMappingCspCsv/Position actual value for aix2
//     TaskSlaveArmControl Inputs/SlaveArmControl.m_slaveRobot.m_slaveArms[1].m_joints[5].m_motorInputs/m_motorEncoder <-> TxPdoMappingCspCsv/Position actual value for aix3
//     TaskSlaveArmControl Inputs/SlaveArmControl.m_slaveRobot.m_slaveArms[1].m_joints[4].m_motorInputs/m_statusWord <-> TxPdoMappingCspCsv/Statusword
//     TaskSlaveArmControl Inputs/SlaveArmControl.m_slaveRobot.m_slaveArms[1].m_joints[5].m_motorInputs/m_statusWord <-> TxPdoMappingCspCsv/Statusword
//     TaskSlaveArmControl Inputs/SlaveArmControl.m_slaveRobot.m_slaveArms[1].m_joints[5].m_motorInputs/m_current <-> TxPdoMappingCspCsv/Torque actual value for aix3
//     TaskSlaveArmControl Inputs/SlaveArmControl.m_slaveRobot.m_slaveArms[1].m_panelInstrumentOnIO <-> TxPdoMappingCspCsv/digital input
//     TaskSlaveArmControl Outputs/SlaveArmControl.m_slaveRobot.m_slaveArms[1].m_joints[4].m_motorOutputs/m_cmdCurrent <-> RxPdoMappingCspCsv/Target Torque value for aix2
//     TaskSlaveArmControl Outputs/SlaveArmControl.m_slaveRobot.m_slaveArms[1].m_joints[5].m_motorOutputs/m_cmdCurrent <-> RxPdoMappingCspCsv/Target Torque value for aix3
//     TaskSlaveArmControl Outputs/SlaveArmControl.m_slaveRobot.m_slaveArms[1].m_joints[4].m_motorOutputs/m_cmdMotorEncoder <-> RxPdoMappingCspCsv/Target position value for aix2
//     TaskSlaveArmControl Outputs/SlaveArmControl.m_slaveRobot.m_slaveArms[1].m_joints[5].m_motorOutputs/m_cmdMotorEncoder <-> RxPdoMappingCspCsv/Target position value for aix3
//     TaskSlaveArmControl Outputs/SlaveArmControl.m_slaveRobot.m_slaveArms[1].m_joints[4].m_motorOutputs/m_controlWord <-> RxPdoMappingCspCsv/Controlword
//     TaskSlaveArmControl Outputs/SlaveArmControl.m_slaveRobot.m_slaveArms[1].m_joints[4].m_motorOutputs/m_opMode <-> RxPdoMappingCspCsv/Modes of operation
//   SlaveController/SlaveController Instance <-> SlaveArm1/SlaveJoint678
//     TaskSlaveArmControl Inputs/SlaveArmControl.m_slaveRobot.m_slaveArms[1].m_joints[6].m_motorInputs/m_current <-> TxPdoMappingCspCsv/Velocity actual value for aix2
//     TaskSlaveArmControl Inputs/SlaveArmControl.m_slaveRobot.m_slaveArms[1].m_joints[6].m_motorInputs/m_linkEncoder <-> TxPdoMappingCspCsv/ENC2 for aix2
//     TaskSlaveArmControl Inputs/SlaveArmControl.m_slaveRobot.m_slaveArms[1].m_joints[7].m_motorInputs/m_linkEncoder <-> TxPdoMappingCspCsv/ENC2 for aix3
//     TaskSlaveArmControl Inputs/SlaveArmControl.m_slaveRobot.m_slaveArms[1].m_joints[8].m_motorInputs/m_linkEncoder <-> TxPdoMappingCspCsv/ENC2 for aix1
//     TaskSlaveArmControl Inputs/SlaveArmControl.m_slaveRobot.m_slaveArms[1].m_joints[6].m_motorInputs/m_motorEncoder <-> TxPdoMappingCspCsv/Position actual value for aix2
//     TaskSlaveArmControl Inputs/SlaveArmControl.m_slaveRobot.m_slaveArms[1].m_joints[7].m_motorInputs/m_motorEncoder <-> TxPdoMappingCspCsv/Position actual value for aix3
//     TaskSlaveArmControl Inputs/SlaveArmControl.m_slaveRobot.m_slaveArms[1].m_joints[6].m_motorInputs/m_statusWord <-> TxPdoMappingCspCsv/Statusword
//     TaskSlaveArmControl Inputs/SlaveArmControl.m_slaveRobot.m_slaveArms[1].m_joints[7].m_motorInputs/m_statusWord <-> TxPdoMappingCspCsv/Statusword
//     TaskSlaveArmControl Inputs/SlaveArmControl.m_slaveRobot.m_slaveArms[1].m_joints[8].m_motorInputs/m_statusWord <-> TxPdoMappingCspCsv/Statusword
//     TaskSlaveArmControl Inputs/SlaveArmControl.m_slaveRobot.m_slaveArms[1].m_joints[7].m_motorInputs/m_current <-> TxPdoMappingCspCsv/Torque actual value for aix3
//     TaskSlaveArmControl Inputs/SlaveArmControl.m_slaveRobot.m_slaveArms[1].m_joints[8].m_motorInputs/m_current <-> TxPdoMappingCspCsv/Torque actual value
//     TaskSlaveArmControl Inputs/SlaveArmControl.m_slaveRobot.m_slaveArms[1].m_joints[8].m_motorInputs/m_motorEncoder <-> TxPdoMappingCspCsv/Position actual value
//     TaskSlaveArmControl Outputs/SlaveArmControl.m_slaveRobot.m_slaveArms[1].m_joints[6].m_motorOutputs/m_cmdCurrent <-> RxPdoMappingCspCsv/Target Torque value for aix2
//     TaskSlaveArmControl Outputs/SlaveArmControl.m_slaveRobot.m_slaveArms[1].m_joints[7].m_motorOutputs/m_cmdCurrent <-> RxPdoMappingCspCsv/Target Torque value for aix3
//     TaskSlaveArmControl Outputs/SlaveArmControl.m_slaveRobot.m_slaveArms[1].m_joints[6].m_motorOutputs/m_cmdMotorEncoder <-> RxPdoMappingCspCsv/Target position value for aix2
//     TaskSlaveArmControl Outputs/SlaveArmControl.m_slaveRobot.m_slaveArms[1].m_joints[7].m_motorOutputs/m_cmdMotorEncoder <-> RxPdoMappingCspCsv/Target position value for aix3
//     TaskSlaveArmControl Outputs/SlaveArmControl.m_slaveRobot.m_slaveArms[1].m_joints[6].m_motorOutputs/m_controlWord <-> RxPdoMappingCspCsv/Controlword
//     TaskSlaveArmControl Outputs/SlaveArmControl.m_slaveRobot.m_slaveArms[1].m_joints[6].m_motorOutputs/m_opMode <-> RxPdoMappingCspCsv/Modes of operation
//     TaskSlaveArmControl Outputs/SlaveArmControl.m_slaveRobot.m_slaveArms[1].m_joints[8].m_motorOutputs/m_cmdCurrent <-> RxPdoMappingCspCsv/Target Torque value
//     TaskSlaveArmControl Outputs/SlaveArmControl.m_slaveRobot.m_slaveArms[1].m_joints[8].m_motorOutputs/m_cmdMotorEncoder <-> RxPdoMappingCspCsv/Target position
//   SlaveController/SlaveController Instance <-> SlaveArm2/SetupJoint12
//     TaskSetupArmControl Inputs/SetupArmControl.m_setupRobot.m_setupArms[2].m_joints[1].m_motorInputs/m_linkEncoder <-> TxPdoMappingCspCsv/ENC2
//     TaskSetupArmControl Inputs/SetupArmControl.m_setupRobot.m_setupArms[2].m_joints[1].m_motorInputs/m_statusWord <-> TxPdoMappingCspCsv/Statusword
//     TaskSetupArmControl Inputs/SetupArmControl.m_setupRobot.m_setupArms[2].m_joints[2].m_motorInputs/m_statusWord <-> TxPdoMappingCspCsv/Statusword
//     TaskSetupArmControl Inputs/SetupArmControl.m_setupRobot.m_setupArms[2].m_joints[2].m_motorInputs/m_linkEncoder <-> TxPdoMappingCspCsv/Torque actual value
//     TaskSetupArmControl Outputs/SetupArmControl.m_setupRobot.m_setupArms[2].m_joints[1].m_motorOutputs/m_controlWord <-> RxPdoMappingCspCsv/Controlword
//   SlaveController/SlaveController Instance <-> SlaveArm2/SetupJoint3
//     TaskSetupArmControl Inputs/SetupArmControl.m_setupRobot.m_setupArms[2].m_joints[3].m_motorInputs/m_current <-> TxPdoMappingCspCsv/Torque actual value
//     TaskSetupArmControl Inputs/SetupArmControl.m_setupRobot.m_setupArms[2].m_joints[3].m_motorInputs/m_linkEncoder <-> TxPdoMappingCspCsv/ENC2
//     TaskSetupArmControl Inputs/SetupArmControl.m_setupRobot.m_setupArms[2].m_joints[3].m_motorInputs/m_motorEncoder <-> TxPdoMappingCspCsv/Position actual value
//     TaskSetupArmControl Inputs/SetupArmControl.m_setupRobot.m_setupArms[2].m_joints[3].m_motorInputs/m_statusWord <-> TxPdoMappingCspCsv/Statusword
//     TaskSetupArmControl Outputs/SetupArmControl.m_setupRobot.m_setupArms[2].m_joints[3].m_motorOutputs/m_cmdCurrent <-> RxPdoMappingCspCsv/Target torque
//     TaskSetupArmControl Outputs/SetupArmControl.m_setupRobot.m_setupArms[2].m_joints[3].m_motorOutputs/m_cmdMotorEncoder <-> RxPdoMappingCspCsv/Target position
//     TaskSetupArmControl Outputs/SetupArmControl.m_setupRobot.m_setupArms[2].m_joints[3].m_motorOutputs/m_controlWord <-> RxPdoMappingCspCsv/Controlword
//     TaskSetupArmControl Outputs/SetupArmControl.m_setupRobot.m_setupArms[2].m_joints[3].m_motorOutputs/m_opMode <-> RxPdoMappingCspCsv/Modes of operation
//   SlaveController/SlaveController Instance <-> SlaveArm2/SetupJoint4
//     TaskSetupArmControl Inputs/SetupArmControl.m_setupRobot.m_setupArms[2].m_joints[4].m_motorInputs/m_current <-> TxPdoMappingCspCsv/Torque actual value
//     TaskSetupArmControl Inputs/SetupArmControl.m_setupRobot.m_setupArms[2].m_joints[4].m_motorInputs/m_motorEncoder <-> TxPdoMappingCspCsv/Position actual value
//     TaskSetupArmControl Inputs/SetupArmControl.m_setupRobot.m_setupArms[2].m_joints[4].m_motorInputs/m_statusWord <-> TxPdoMappingCspCsv/Statusword
//     TaskSetupArmControl Outputs/SetupArmControl.m_setupRobot.m_setupArms[2].m_joints[4].m_motorOutputs/m_cmdCurrent <-> RxPdoMappingCspCsv/Target torque
//     TaskSetupArmControl Outputs/SetupArmControl.m_setupRobot.m_setupArms[2].m_joints[4].m_motorOutputs/m_cmdMotorEncoder <-> RxPdoMappingCspCsv/Target position
//     TaskSetupArmControl Outputs/SetupArmControl.m_setupRobot.m_setupArms[2].m_joints[4].m_motorOutputs/m_controlWord <-> RxPdoMappingCspCsv/Controlword
//     TaskSetupArmControl Outputs/SetupArmControl.m_setupRobot.m_setupArms[2].m_joints[4].m_motorOutputs/m_opMode <-> RxPdoMappingCspCsv/Modes of operation
//   SlaveController/SlaveController Instance <-> SlaveArm2/SetupJoint5
//     TaskSetupArmControl Inputs/SetupArmControl.m_setupRobot.m_setupArms[2].m_joints[4].m_motorInputs/m_linkEncoder <-> TxPdoMappingCspCsv/ENC2
//     TaskSetupArmControl Inputs/SetupArmControl.m_setupRobot.m_setupArms[2].m_joints[5].m_motorInputs/m_current <-> TxPdoMappingCspCsv/Torque actual value
//     TaskSetupArmControl Inputs/SetupArmControl.m_setupRobot.m_setupArms[2].m_joints[5].m_motorInputs/m_linkEncoder <-> TxPdoMappingCspCsv/analog input
//     TaskSetupArmControl Inputs/SetupArmControl.m_setupRobot.m_setupArms[2].m_joints[5].m_motorInputs/m_motorEncoder <-> TxPdoMappingCspCsv/Position actual value
//     TaskSetupArmControl Inputs/SetupArmControl.m_setupRobot.m_setupArms[2].m_joints[5].m_motorInputs/m_statusWord <-> TxPdoMappingCspCsv/Statusword
//     TaskSetupArmControl Outputs/SetupArmControl.m_setupRobot.m_setupArms[2].m_joints[5].m_motorOutputs/m_cmdCurrent <-> RxPdoMappingCspCsv/Target torque
//     TaskSetupArmControl Outputs/SetupArmControl.m_setupRobot.m_setupArms[2].m_joints[5].m_motorOutputs/m_cmdMotorEncoder <-> RxPdoMappingCspCsv/Target position
//     TaskSetupArmControl Outputs/SetupArmControl.m_setupRobot.m_setupArms[2].m_joints[5].m_motorOutputs/m_controlWord <-> RxPdoMappingCspCsv/Controlword
//     TaskSetupArmControl Outputs/SetupArmControl.m_setupRobot.m_setupArms[2].m_joints[5].m_motorOutputs/m_opMode <-> RxPdoMappingCspCsv/Modes of operation
//   SlaveController/SlaveController Instance <-> SlaveArm2/SlaveJoint1
//     TaskSlaveArmControl Inputs/SlaveArmControl.m_slaveRobot.m_slaveArms[2].m_joints[1].m_motorInputs/m_current <-> TxPdoMappingCspCsv/Torque actual value
//     TaskSlaveArmControl Inputs/SlaveArmControl.m_slaveRobot.m_slaveArms[2].m_joints[1].m_motorInputs/m_linkEncoder <-> TxPdoMappingCspCsv/ENC2
//     TaskSlaveArmControl Inputs/SlaveArmControl.m_slaveRobot.m_slaveArms[2].m_joints[1].m_motorInputs/m_motorEncoder <-> TxPdoMappingCspCsv/Position actual value
//     TaskSlaveArmControl Inputs/SlaveArmControl.m_slaveRobot.m_slaveArms[2].m_joints[1].m_motorInputs/m_statusWord <-> TxPdoMappingCspCsv/Statusword
//     TaskSlaveArmControl Outputs/SlaveArmControl.m_slaveRobot.m_slaveArms[2].m_joints[1].m_motorOutputs/m_cmdCurrent <-> RxPdoMappingCspCsv/Target torque
//     TaskSlaveArmControl Outputs/SlaveArmControl.m_slaveRobot.m_slaveArms[2].m_joints[1].m_motorOutputs/m_cmdMotorEncoder <-> RxPdoMappingCspCsv/Target position
//     TaskSlaveArmControl Outputs/SlaveArmControl.m_slaveRobot.m_slaveArms[2].m_joints[1].m_motorOutputs/m_controlWord <-> RxPdoMappingCspCsv/Controlword
//     TaskSlaveArmControl Outputs/SlaveArmControl.m_slaveRobot.m_slaveArms[2].m_joints[1].m_motorOutputs/m_opMode <-> RxPdoMappingCspCsv/Modes of operation
//   SlaveController/SlaveController Instance <-> SlaveArm2/SlaveJoint2
//     TaskCartControl Inputs/CartControl.m_cartRobot.m_slaveCart.m_carRotaOverhangIO[2] <-> TxPdoMappingCspCsv/digital input
//     TaskSetupArmControl Outputs/SetupArmControl.m_setupRobot.m_setupArms[2].m_lightIO <-> RxPdoMappingCspCsv/Target velocity
//     TaskSlaveArmControl Inputs/SlaveArmControl.m_slaveRobot.m_slaveArms[2].m_joints[2].m_motorInputs/m_current <-> TxPdoMappingCspCsv/Torque actual value
//     TaskSlaveArmControl Inputs/SlaveArmControl.m_slaveRobot.m_slaveArms[2].m_joints[2].m_motorInputs/m_linkEncoder <-> TxPdoMappingCspCsv/ENC2
//     TaskSlaveArmControl Inputs/SlaveArmControl.m_slaveRobot.m_slaveArms[2].m_joints[2].m_motorInputs/m_motorEncoder <-> TxPdoMappingCspCsv/Position actual value
//     TaskSlaveArmControl Inputs/SlaveArmControl.m_slaveRobot.m_slaveArms[2].m_joints[2].m_motorInputs/m_statusWord <-> TxPdoMappingCspCsv/Statusword
//     TaskSlaveArmControl Outputs/SlaveArmControl.m_slaveRobot.m_slaveArms[2].m_joints[2].m_motorOutputs/m_cmdCurrent <-> RxPdoMappingCspCsv/Target torque
//     TaskSlaveArmControl Outputs/SlaveArmControl.m_slaveRobot.m_slaveArms[2].m_joints[2].m_motorOutputs/m_cmdMotorEncoder <-> RxPdoMappingCspCsv/Target position
//     TaskSlaveArmControl Outputs/SlaveArmControl.m_slaveRobot.m_slaveArms[2].m_joints[2].m_motorOutputs/m_controlWord <-> RxPdoMappingCspCsv/Controlword
//     TaskSlaveArmControl Outputs/SlaveArmControl.m_slaveRobot.m_slaveArms[2].m_joints[2].m_motorOutputs/m_opMode <-> RxPdoMappingCspCsv/Modes of operation
//   SlaveController/SlaveController Instance <-> SlaveArm2/SlaveJoint3
//     TaskCartControl Inputs/CartControl.m_cartRobot.m_slaveCart.m_trocarIO[2] <-> TxPdoMappingCspCsv/digital input
//     TaskSetupArmControl Inputs/SetupArmControl.m_setupRobot.m_setupArms[2].m_adjustIO <-> TxPdoMappingCspCsv/digital input
//     TaskSlaveArmControl Inputs/SlaveArmControl.m_slaveRobot.m_slaveArms[2].m_adjustIO <-> TxPdoMappingCspCsv/digital input
//     TaskSlaveArmControl Inputs/SlaveArmControl.m_slaveRobot.m_slaveArms[2].m_joints[3].m_motorInputs/m_current <-> TxPdoMappingCspCsv/Torque actual value
//     TaskSlaveArmControl Inputs/SlaveArmControl.m_slaveRobot.m_slaveArms[2].m_joints[3].m_motorInputs/m_linkEncoder <-> TxPdoMappingCspCsv/ENC2 for aix1
//     TaskSlaveArmControl Inputs/SlaveArmControl.m_slaveRobot.m_slaveArms[2].m_joints[3].m_motorInputs/m_motorEncoder <-> TxPdoMappingCspCsv/Position actual value
//     TaskSlaveArmControl Inputs/SlaveArmControl.m_slaveRobot.m_slaveArms[2].m_joints[3].m_motorInputs/m_statusWord <-> TxPdoMappingCspCsv/Statusword
//     TaskSlaveArmControl Outputs/SlaveArmControl.m_slaveRobot.m_slaveArms[2].m_joints[3].m_motorOutputs/m_cmdCurrent <-> RxPdoMappingCspCsv/Target Torque value
//     TaskSlaveArmControl Outputs/SlaveArmControl.m_slaveRobot.m_slaveArms[2].m_joints[3].m_motorOutputs/m_cmdMotorEncoder <-> RxPdoMappingCspCsv/Target position
//     TaskSlaveArmControl Outputs/SlaveArmControl.m_slaveRobot.m_slaveArms[2].m_joints[3].m_motorOutputs/m_controlWord <-> RxPdoMappingCspCsv/Controlword
//     TaskSlaveArmControl Outputs/SlaveArmControl.m_slaveRobot.m_slaveArms[2].m_joints[3].m_motorOutputs/m_opMode <-> RxPdoMappingCspCsv/Modes of operation
//   SlaveController/SlaveController Instance <-> SlaveArm2/SlaveJoint45
//     TaskSlaveArmControl Inputs/SlaveArmControl.m_slaveRobot.m_slaveArms[2].m_joints[4].m_motorInputs/m_current <-> TxPdoMappingCspCsv/Velocity actual value for aix2
//     TaskSlaveArmControl Inputs/SlaveArmControl.m_slaveRobot.m_slaveArms[2].m_joints[4].m_motorInputs/m_linkEncoder <-> TxPdoMappingCspCsv/ENC2 for aix2
//     TaskSlaveArmControl Inputs/SlaveArmControl.m_slaveRobot.m_slaveArms[2].m_joints[5].m_motorInputs/m_linkEncoder <-> TxPdoMappingCspCsv/ENC2 for aix3
//     TaskSlaveArmControl Inputs/SlaveArmControl.m_slaveRobot.m_slaveArms[2].m_joints[4].m_motorInputs/m_motorEncoder <-> TxPdoMappingCspCsv/Position actual value for aix2
//     TaskSlaveArmControl Inputs/SlaveArmControl.m_slaveRobot.m_slaveArms[2].m_joints[5].m_motorInputs/m_motorEncoder <-> TxPdoMappingCspCsv/Position actual value for aix3
//     TaskSlaveArmControl Inputs/SlaveArmControl.m_slaveRobot.m_slaveArms[2].m_joints[4].m_motorInputs/m_statusWord <-> TxPdoMappingCspCsv/Statusword
//     TaskSlaveArmControl Inputs/SlaveArmControl.m_slaveRobot.m_slaveArms[2].m_joints[5].m_motorInputs/m_statusWord <-> TxPdoMappingCspCsv/Statusword
//     TaskSlaveArmControl Inputs/SlaveArmControl.m_slaveRobot.m_slaveArms[2].m_joints[5].m_motorInputs/m_current <-> TxPdoMappingCspCsv/Torque actual value for aix3
//     TaskSlaveArmControl Inputs/SlaveArmControl.m_slaveRobot.m_slaveArms[2].m_panelInstrumentOnIO <-> TxPdoMappingCspCsv/digital input
//     TaskSlaveArmControl Outputs/SlaveArmControl.m_slaveRobot.m_slaveArms[2].m_joints[4].m_motorOutputs/m_cmdCurrent <-> RxPdoMappingCspCsv/Target Torque value for aix2
//     TaskSlaveArmControl Outputs/SlaveArmControl.m_slaveRobot.m_slaveArms[2].m_joints[5].m_motorOutputs/m_cmdCurrent <-> RxPdoMappingCspCsv/Target Torque value for aix3
//     TaskSlaveArmControl Outputs/SlaveArmControl.m_slaveRobot.m_slaveArms[2].m_joints[4].m_motorOutputs/m_cmdMotorEncoder <-> RxPdoMappingCspCsv/Target position value for aix2
//     TaskSlaveArmControl Outputs/SlaveArmControl.m_slaveRobot.m_slaveArms[2].m_joints[5].m_motorOutputs/m_cmdMotorEncoder <-> RxPdoMappingCspCsv/Target position value for aix3
//     TaskSlaveArmControl Outputs/SlaveArmControl.m_slaveRobot.m_slaveArms[2].m_joints[4].m_motorOutputs/m_controlWord <-> RxPdoMappingCspCsv/Controlword
//     TaskSlaveArmControl Outputs/SlaveArmControl.m_slaveRobot.m_slaveArms[2].m_joints[4].m_motorOutputs/m_opMode <-> RxPdoMappingCspCsv/Modes of operation
//   SlaveController/SlaveController Instance <-> SlaveArm2/SlaveJoint678
//     TaskSlaveArmControl Inputs/SlaveArmControl.m_slaveRobot.m_slaveArms[2].m_joints[6].m_motorInputs/m_current <-> TxPdoMappingCspCsv/Velocity actual value for aix2
//     TaskSlaveArmControl Inputs/SlaveArmControl.m_slaveRobot.m_slaveArms[2].m_joints[6].m_motorInputs/m_linkEncoder <-> TxPdoMappingCspCsv/ENC2 for aix2
//     TaskSlaveArmControl Inputs/SlaveArmControl.m_slaveRobot.m_slaveArms[2].m_joints[7].m_motorInputs/m_linkEncoder <-> TxPdoMappingCspCsv/ENC2 for aix3
//     TaskSlaveArmControl Inputs/SlaveArmControl.m_slaveRobot.m_slaveArms[2].m_joints[8].m_motorInputs/m_linkEncoder <-> TxPdoMappingCspCsv/ENC2 for aix1
//     TaskSlaveArmControl Inputs/SlaveArmControl.m_slaveRobot.m_slaveArms[2].m_joints[6].m_motorInputs/m_motorEncoder <-> TxPdoMappingCspCsv/Position actual value for aix2
//     TaskSlaveArmControl Inputs/SlaveArmControl.m_slaveRobot.m_slaveArms[2].m_joints[7].m_motorInputs/m_motorEncoder <-> TxPdoMappingCspCsv/Position actual value for aix3
//     TaskSlaveArmControl Inputs/SlaveArmControl.m_slaveRobot.m_slaveArms[2].m_joints[6].m_motorInputs/m_statusWord <-> TxPdoMappingCspCsv/Statusword
//     TaskSlaveArmControl Inputs/SlaveArmControl.m_slaveRobot.m_slaveArms[2].m_joints[7].m_motorInputs/m_statusWord <-> TxPdoMappingCspCsv/Statusword
//     TaskSlaveArmControl Inputs/SlaveArmControl.m_slaveRobot.m_slaveArms[2].m_joints[8].m_motorInputs/m_statusWord <-> TxPdoMappingCspCsv/Statusword
//     TaskSlaveArmControl Inputs/SlaveArmControl.m_slaveRobot.m_slaveArms[2].m_joints[7].m_motorInputs/m_current <-> TxPdoMappingCspCsv/Torque actual value for aix3
//     TaskSlaveArmControl Inputs/SlaveArmControl.m_slaveRobot.m_slaveArms[2].m_joints[8].m_motorInputs/m_current <-> TxPdoMappingCspCsv/Torque actual value
//     TaskSlaveArmControl Inputs/SlaveArmControl.m_slaveRobot.m_slaveArms[2].m_joints[8].m_motorInputs/m_motorEncoder <-> TxPdoMappingCspCsv/Position actual value
//     TaskSlaveArmControl Outputs/SlaveArmControl.m_slaveRobot.m_slaveArms[2].m_joints[6].m_motorOutputs/m_cmdCurrent <-> RxPdoMappingCspCsv/Target Torque value for aix2
//     TaskSlaveArmControl Outputs/SlaveArmControl.m_slaveRobot.m_slaveArms[2].m_joints[7].m_motorOutputs/m_cmdCurrent <-> RxPdoMappingCspCsv/Target Torque value for aix3
//     TaskSlaveArmControl Outputs/SlaveArmControl.m_slaveRobot.m_slaveArms[2].m_joints[6].m_motorOutputs/m_cmdMotorEncoder <-> RxPdoMappingCspCsv/Target position value for aix2
//     TaskSlaveArmControl Outputs/SlaveArmControl.m_slaveRobot.m_slaveArms[2].m_joints[7].m_motorOutputs/m_cmdMotorEncoder <-> RxPdoMappingCspCsv/Target position value for aix3
//     TaskSlaveArmControl Outputs/SlaveArmControl.m_slaveRobot.m_slaveArms[2].m_joints[6].m_motorOutputs/m_controlWord <-> RxPdoMappingCspCsv/Controlword
//     TaskSlaveArmControl Outputs/SlaveArmControl.m_slaveRobot.m_slaveArms[2].m_joints[6].m_motorOutputs/m_opMode <-> RxPdoMappingCspCsv/Modes of operation
//     TaskSlaveArmControl Outputs/SlaveArmControl.m_slaveRobot.m_slaveArms[2].m_joints[8].m_motorOutputs/m_cmdCurrent <-> RxPdoMappingCspCsv/Target Torque value
//     TaskSlaveArmControl Outputs/SlaveArmControl.m_slaveRobot.m_slaveArms[2].m_joints[8].m_motorOutputs/m_cmdMotorEncoder <-> RxPdoMappingCspCsv/Target position
//   SlaveController/SlaveController Instance <-> SlaveArm3/SetupJoint12
//     TaskSetupArmControl Inputs/SetupArmControl.m_setupRobot.m_setupArms[3].m_joints[1].m_motorInputs/m_linkEncoder <-> TxPdoMappingCspCsv/ENC2
//     TaskSetupArmControl Inputs/SetupArmControl.m_setupRobot.m_setupArms[3].m_joints[1].m_motorInputs/m_statusWord <-> TxPdoMappingCspCsv/Statusword
//     TaskSetupArmControl Inputs/SetupArmControl.m_setupRobot.m_setupArms[3].m_joints[2].m_motorInputs/m_statusWord <-> TxPdoMappingCspCsv/Statusword
//     TaskSetupArmControl Inputs/SetupArmControl.m_setupRobot.m_setupArms[3].m_joints[2].m_motorInputs/m_linkEncoder <-> TxPdoMappingCspCsv/Torque actual value
//     TaskSetupArmControl Outputs/SetupArmControl.m_setupRobot.m_setupArms[3].m_joints[1].m_motorOutputs/m_controlWord <-> RxPdoMappingCspCsv/Controlword
//   SlaveController/SlaveController Instance <-> SlaveArm3/SetupJoint3
//     TaskSetupArmControl Inputs/SetupArmControl.m_setupRobot.m_setupArms[3].m_joints[3].m_motorInputs/m_current <-> TxPdoMappingCspCsv/Torque actual value
//     TaskSetupArmControl Inputs/SetupArmControl.m_setupRobot.m_setupArms[3].m_joints[3].m_motorInputs/m_linkEncoder <-> TxPdoMappingCspCsv/ENC2
//     TaskSetupArmControl Inputs/SetupArmControl.m_setupRobot.m_setupArms[3].m_joints[3].m_motorInputs/m_motorEncoder <-> TxPdoMappingCspCsv/Position actual value
//     TaskSetupArmControl Inputs/SetupArmControl.m_setupRobot.m_setupArms[3].m_joints[3].m_motorInputs/m_statusWord <-> TxPdoMappingCspCsv/Statusword
//     TaskSetupArmControl Outputs/SetupArmControl.m_setupRobot.m_setupArms[3].m_joints[3].m_motorOutputs/m_cmdCurrent <-> RxPdoMappingCspCsv/Target torque
//     TaskSetupArmControl Outputs/SetupArmControl.m_setupRobot.m_setupArms[3].m_joints[3].m_motorOutputs/m_cmdMotorEncoder <-> RxPdoMappingCspCsv/Target position
//     TaskSetupArmControl Outputs/SetupArmControl.m_setupRobot.m_setupArms[3].m_joints[3].m_motorOutputs/m_controlWord <-> RxPdoMappingCspCsv/Controlword
//     TaskSetupArmControl Outputs/SetupArmControl.m_setupRobot.m_setupArms[3].m_joints[3].m_motorOutputs/m_opMode <-> RxPdoMappingCspCsv/Modes of operation
//   SlaveController/SlaveController Instance <-> SlaveArm3/SetupJoint4
//     TaskSetupArmControl Inputs/SetupArmControl.m_setupRobot.m_setupArms[3].m_joints[4].m_motorInputs/m_current <-> TxPdoMappingCspCsv/Torque actual value
//     TaskSetupArmControl Inputs/SetupArmControl.m_setupRobot.m_setupArms[3].m_joints[4].m_motorInputs/m_motorEncoder <-> TxPdoMappingCspCsv/Position actual value
//     TaskSetupArmControl Inputs/SetupArmControl.m_setupRobot.m_setupArms[3].m_joints[4].m_motorInputs/m_statusWord <-> TxPdoMappingCspCsv/Statusword
//     TaskSetupArmControl Outputs/SetupArmControl.m_setupRobot.m_setupArms[3].m_joints[4].m_motorOutputs/m_cmdCurrent <-> RxPdoMappingCspCsv/Target torque
//     TaskSetupArmControl Outputs/SetupArmControl.m_setupRobot.m_setupArms[3].m_joints[4].m_motorOutputs/m_cmdMotorEncoder <-> RxPdoMappingCspCsv/Target position
//     TaskSetupArmControl Outputs/SetupArmControl.m_setupRobot.m_setupArms[3].m_joints[4].m_motorOutputs/m_controlWord <-> RxPdoMappingCspCsv/Controlword
//     TaskSetupArmControl Outputs/SetupArmControl.m_setupRobot.m_setupArms[3].m_joints[4].m_motorOutputs/m_opMode <-> RxPdoMappingCspCsv/Modes of operation
//   SlaveController/SlaveController Instance <-> SlaveArm3/SetupJoint5
//     TaskSetupArmControl Inputs/SetupArmControl.m_setupRobot.m_setupArms[3].m_joints[4].m_motorInputs/m_linkEncoder <-> TxPdoMappingCspCsv/ENC2
//     TaskSetupArmControl Inputs/SetupArmControl.m_setupRobot.m_setupArms[3].m_joints[5].m_motorInputs/m_current <-> TxPdoMappingCspCsv/Torque actual value
//     TaskSetupArmControl Inputs/SetupArmControl.m_setupRobot.m_setupArms[3].m_joints[5].m_motorInputs/m_linkEncoder <-> TxPdoMappingCspCsv/analog input
//     TaskSetupArmControl Inputs/SetupArmControl.m_setupRobot.m_setupArms[3].m_joints[5].m_motorInputs/m_motorEncoder <-> TxPdoMappingCspCsv/Position actual value
//     TaskSetupArmControl Inputs/SetupArmControl.m_setupRobot.m_setupArms[3].m_joints[5].m_motorInputs/m_statusWord <-> TxPdoMappingCspCsv/Statusword
//     TaskSetupArmControl Outputs/SetupArmControl.m_setupRobot.m_setupArms[3].m_joints[5].m_motorOutputs/m_cmdCurrent <-> RxPdoMappingCspCsv/Target torque
//     TaskSetupArmControl Outputs/SetupArmControl.m_setupRobot.m_setupArms[3].m_joints[5].m_motorOutputs/m_cmdMotorEncoder <-> RxPdoMappingCspCsv/Target position
//     TaskSetupArmControl Outputs/SetupArmControl.m_setupRobot.m_setupArms[3].m_joints[5].m_motorOutputs/m_controlWord <-> RxPdoMappingCspCsv/Controlword
//     TaskSetupArmControl Outputs/SetupArmControl.m_setupRobot.m_setupArms[3].m_joints[5].m_motorOutputs/m_opMode <-> RxPdoMappingCspCsv/Modes of operation
//   SlaveController/SlaveController Instance <-> SlaveArm3/SlaveJoint1
//     TaskSlaveArmControl Inputs/SlaveArmControl.m_slaveRobot.m_slaveArms[3].m_joints[1].m_motorInputs/m_current <-> TxPdoMappingCspCsv/Torque actual value
//     TaskSlaveArmControl Inputs/SlaveArmControl.m_slaveRobot.m_slaveArms[3].m_joints[1].m_motorInputs/m_linkEncoder <-> TxPdoMappingCspCsv/ENC2
//     TaskSlaveArmControl Inputs/SlaveArmControl.m_slaveRobot.m_slaveArms[3].m_joints[1].m_motorInputs/m_motorEncoder <-> TxPdoMappingCspCsv/Position actual value
//     TaskSlaveArmControl Inputs/SlaveArmControl.m_slaveRobot.m_slaveArms[3].m_joints[1].m_motorInputs/m_statusWord <-> TxPdoMappingCspCsv/Statusword
//     TaskSlaveArmControl Outputs/SlaveArmControl.m_slaveRobot.m_slaveArms[3].m_joints[1].m_motorOutputs/m_cmdCurrent <-> RxPdoMappingCspCsv/Target torque
//     TaskSlaveArmControl Outputs/SlaveArmControl.m_slaveRobot.m_slaveArms[3].m_joints[1].m_motorOutputs/m_cmdMotorEncoder <-> RxPdoMappingCspCsv/Target position
//     TaskSlaveArmControl Outputs/SlaveArmControl.m_slaveRobot.m_slaveArms[3].m_joints[1].m_motorOutputs/m_controlWord <-> RxPdoMappingCspCsv/Controlword
//     TaskSlaveArmControl Outputs/SlaveArmControl.m_slaveRobot.m_slaveArms[3].m_joints[1].m_motorOutputs/m_opMode <-> RxPdoMappingCspCsv/Modes of operation
//   SlaveController/SlaveController Instance <-> SlaveArm3/SlaveJoint2
//     TaskCartControl Inputs/CartControl.m_cartRobot.m_slaveCart.m_carRotaOverhangIO[3] <-> TxPdoMappingCspCsv/digital input
//     TaskSetupArmControl Outputs/SetupArmControl.m_setupRobot.m_setupArms[3].m_lightIO <-> RxPdoMappingCspCsv/Target velocity
//     TaskSlaveArmControl Inputs/SlaveArmControl.m_slaveRobot.m_slaveArms[3].m_joints[2].m_motorInputs/m_current <-> TxPdoMappingCspCsv/Torque actual value
//     TaskSlaveArmControl Inputs/SlaveArmControl.m_slaveRobot.m_slaveArms[3].m_joints[2].m_motorInputs/m_linkEncoder <-> TxPdoMappingCspCsv/ENC2
//     TaskSlaveArmControl Inputs/SlaveArmControl.m_slaveRobot.m_slaveArms[3].m_joints[2].m_motorInputs/m_motorEncoder <-> TxPdoMappingCspCsv/Position actual value
//     TaskSlaveArmControl Inputs/SlaveArmControl.m_slaveRobot.m_slaveArms[3].m_joints[2].m_motorInputs/m_statusWord <-> TxPdoMappingCspCsv/Statusword
//     TaskSlaveArmControl Outputs/SlaveArmControl.m_slaveRobot.m_slaveArms[3].m_joints[2].m_motorOutputs/m_cmdCurrent <-> RxPdoMappingCspCsv/Target torque
//     TaskSlaveArmControl Outputs/SlaveArmControl.m_slaveRobot.m_slaveArms[3].m_joints[2].m_motorOutputs/m_cmdMotorEncoder <-> RxPdoMappingCspCsv/Target position
//     TaskSlaveArmControl Outputs/SlaveArmControl.m_slaveRobot.m_slaveArms[3].m_joints[2].m_motorOutputs/m_controlWord <-> RxPdoMappingCspCsv/Controlword
//     TaskSlaveArmControl Outputs/SlaveArmControl.m_slaveRobot.m_slaveArms[3].m_joints[2].m_motorOutputs/m_opMode <-> RxPdoMappingCspCsv/Modes of operation
//   SlaveController/SlaveController Instance <-> SlaveArm3/SlaveJoint3
//     TaskCartControl Inputs/CartControl.m_cartRobot.m_slaveCart.m_trocarIO[3] <-> TxPdoMappingCspCsv/digital input
//     TaskSetupArmControl Inputs/SetupArmControl.m_setupRobot.m_setupArms[3].m_adjustIO <-> TxPdoMappingCspCsv/digital input
//     TaskSlaveArmControl Inputs/SlaveArmControl.m_slaveRobot.m_slaveArms[3].m_adjustIO <-> TxPdoMappingCspCsv/digital input
//     TaskSlaveArmControl Inputs/SlaveArmControl.m_slaveRobot.m_slaveArms[3].m_joints[3].m_motorInputs/m_current <-> TxPdoMappingCspCsv/Torque actual value
//     TaskSlaveArmControl Inputs/SlaveArmControl.m_slaveRobot.m_slaveArms[3].m_joints[3].m_motorInputs/m_linkEncoder <-> TxPdoMappingCspCsv/ENC2 for aix1
//     TaskSlaveArmControl Inputs/SlaveArmControl.m_slaveRobot.m_slaveArms[3].m_joints[3].m_motorInputs/m_motorEncoder <-> TxPdoMappingCspCsv/Position actual value
//     TaskSlaveArmControl Inputs/SlaveArmControl.m_slaveRobot.m_slaveArms[3].m_joints[3].m_motorInputs/m_statusWord <-> TxPdoMappingCspCsv/Statusword
//     TaskSlaveArmControl Outputs/SlaveArmControl.m_slaveRobot.m_slaveArms[3].m_joints[3].m_motorOutputs/m_cmdCurrent <-> RxPdoMappingCspCsv/Target Torque value
//     TaskSlaveArmControl Outputs/SlaveArmControl.m_slaveRobot.m_slaveArms[3].m_joints[3].m_motorOutputs/m_cmdMotorEncoder <-> RxPdoMappingCspCsv/Target position
//     TaskSlaveArmControl Outputs/SlaveArmControl.m_slaveRobot.m_slaveArms[3].m_joints[3].m_motorOutputs/m_controlWord <-> RxPdoMappingCspCsv/Controlword
//     TaskSlaveArmControl Outputs/SlaveArmControl.m_slaveRobot.m_slaveArms[3].m_joints[3].m_motorOutputs/m_opMode <-> RxPdoMappingCspCsv/Modes of operation
//   SlaveController/SlaveController Instance <-> SlaveArm3/SlaveJoint45
//     TaskSlaveArmControl Inputs/SlaveArmControl.m_slaveRobot.m_slaveArms[3].m_joints[4].m_motorInputs/m_current <-> TxPdoMappingCspCsv/Velocity actual value for aix2
//     TaskSlaveArmControl Inputs/SlaveArmControl.m_slaveRobot.m_slaveArms[3].m_joints[4].m_motorInputs/m_linkEncoder <-> TxPdoMappingCspCsv/ENC2 for aix2
//     TaskSlaveArmControl Inputs/SlaveArmControl.m_slaveRobot.m_slaveArms[3].m_joints[5].m_motorInputs/m_linkEncoder <-> TxPdoMappingCspCsv/ENC2 for aix3
//     TaskSlaveArmControl Inputs/SlaveArmControl.m_slaveRobot.m_slaveArms[3].m_joints[4].m_motorInputs/m_motorEncoder <-> TxPdoMappingCspCsv/Position actual value for aix2
//     TaskSlaveArmControl Inputs/SlaveArmControl.m_slaveRobot.m_slaveArms[3].m_joints[5].m_motorInputs/m_motorEncoder <-> TxPdoMappingCspCsv/Position actual value for aix3
//     TaskSlaveArmControl Inputs/SlaveArmControl.m_slaveRobot.m_slaveArms[3].m_joints[4].m_motorInputs/m_statusWord <-> TxPdoMappingCspCsv/Statusword
//     TaskSlaveArmControl Inputs/SlaveArmControl.m_slaveRobot.m_slaveArms[3].m_joints[5].m_motorInputs/m_statusWord <-> TxPdoMappingCspCsv/Statusword
//     TaskSlaveArmControl Inputs/SlaveArmControl.m_slaveRobot.m_slaveArms[3].m_joints[5].m_motorInputs/m_current <-> TxPdoMappingCspCsv/Torque actual value for aix3
//     TaskSlaveArmControl Inputs/SlaveArmControl.m_slaveRobot.m_slaveArms[3].m_panelInstrumentOnIO <-> TxPdoMappingCspCsv/digital input
//     TaskSlaveArmControl Outputs/SlaveArmControl.m_slaveRobot.m_slaveArms[3].m_joints[4].m_motorOutputs/m_cmdCurrent <-> RxPdoMappingCspCsv/Target Torque value for aix2
//     TaskSlaveArmControl Outputs/SlaveArmControl.m_slaveRobot.m_slaveArms[3].m_joints[5].m_motorOutputs/m_cmdCurrent <-> RxPdoMappingCspCsv/Target Torque value for aix3
//     TaskSlaveArmControl Outputs/SlaveArmControl.m_slaveRobot.m_slaveArms[3].m_joints[4].m_motorOutputs/m_cmdMotorEncoder <-> RxPdoMappingCspCsv/Target position value for aix2
//     TaskSlaveArmControl Outputs/SlaveArmControl.m_slaveRobot.m_slaveArms[3].m_joints[5].m_motorOutputs/m_cmdMotorEncoder <-> RxPdoMappingCspCsv/Target position value for aix3
//     TaskSlaveArmControl Outputs/SlaveArmControl.m_slaveRobot.m_slaveArms[3].m_joints[4].m_motorOutputs/m_controlWord <-> RxPdoMappingCspCsv/Controlword
//     TaskSlaveArmControl Outputs/SlaveArmControl.m_slaveRobot.m_slaveArms[3].m_joints[4].m_motorOutputs/m_opMode <-> RxPdoMappingCspCsv/Modes of operation
//   SlaveController/SlaveController Instance <-> SlaveArm3/SlaveJoint678
//     TaskSlaveArmControl Inputs/SlaveArmControl.m_slaveRobot.m_slaveArms[3].m_joints[6].m_motorInputs/m_current <-> TxPdoMappingCspCsv/Velocity actual value for aix2
//     TaskSlaveArmControl Inputs/SlaveArmControl.m_slaveRobot.m_slaveArms[3].m_joints[6].m_motorInputs/m_linkEncoder <-> TxPdoMappingCspCsv/ENC2 for aix2
//     TaskSlaveArmControl Inputs/SlaveArmControl.m_slaveRobot.m_slaveArms[3].m_joints[7].m_motorInputs/m_linkEncoder <-> TxPdoMappingCspCsv/ENC2 for aix3
//     TaskSlaveArmControl Inputs/SlaveArmControl.m_slaveRobot.m_slaveArms[3].m_joints[8].m_motorInputs/m_linkEncoder <-> TxPdoMappingCspCsv/ENC2 for aix1
//     TaskSlaveArmControl Inputs/SlaveArmControl.m_slaveRobot.m_slaveArms[3].m_joints[6].m_motorInputs/m_motorEncoder <-> TxPdoMappingCspCsv/Position actual value for aix2
//     TaskSlaveArmControl Inputs/SlaveArmControl.m_slaveRobot.m_slaveArms[3].m_joints[7].m_motorInputs/m_motorEncoder <-> TxPdoMappingCspCsv/Position actual value for aix3
//     TaskSlaveArmControl Inputs/SlaveArmControl.m_slaveRobot.m_slaveArms[3].m_joints[6].m_motorInputs/m_statusWord <-> TxPdoMappingCspCsv/Statusword
//     TaskSlaveArmControl Inputs/SlaveArmControl.m_slaveRobot.m_slaveArms[3].m_joints[7].m_motorInputs/m_statusWord <-> TxPdoMappingCspCsv/Statusword
//     TaskSlaveArmControl Inputs/SlaveArmControl.m_slaveRobot.m_slaveArms[3].m_joints[8].m_motorInputs/m_statusWord <-> TxPdoMappingCspCsv/Statusword
//     TaskSlaveArmControl Inputs/SlaveArmControl.m_slaveRobot.m_slaveArms[3].m_joints[7].m_motorInputs/m_current <-> TxPdoMappingCspCsv/Torque actual value for aix3
//     TaskSlaveArmControl Inputs/SlaveArmControl.m_slaveRobot.m_slaveArms[3].m_joints[8].m_motorInputs/m_current <-> TxPdoMappingCspCsv/Torque actual value
//     TaskSlaveArmControl Inputs/SlaveArmControl.m_slaveRobot.m_slaveArms[3].m_joints[8].m_motorInputs/m_motorEncoder <-> TxPdoMappingCspCsv/Position actual value
//     TaskSlaveArmControl Outputs/SlaveArmControl.m_slaveRobot.m_slaveArms[3].m_joints[6].m_motorOutputs/m_cmdCurrent <-> RxPdoMappingCspCsv/Target Torque value for aix2
//     TaskSlaveArmControl Outputs/SlaveArmControl.m_slaveRobot.m_slaveArms[3].m_joints[7].m_motorOutputs/m_cmdCurrent <-> RxPdoMappingCspCsv/Target Torque value for aix3
//     TaskSlaveArmControl Outputs/SlaveArmControl.m_slaveRobot.m_slaveArms[3].m_joints[6].m_motorOutputs/m_cmdMotorEncoder <-> RxPdoMappingCspCsv/Target position value for aix2
//     TaskSlaveArmControl Outputs/SlaveArmControl.m_slaveRobot.m_slaveArms[3].m_joints[7].m_motorOutputs/m_cmdMotorEncoder <-> RxPdoMappingCspCsv/Target position value for aix3
//     TaskSlaveArmControl Outputs/SlaveArmControl.m_slaveRobot.m_slaveArms[3].m_joints[6].m_motorOutputs/m_controlWord <-> RxPdoMappingCspCsv/Controlword
//     TaskSlaveArmControl Outputs/SlaveArmControl.m_slaveRobot.m_slaveArms[3].m_joints[6].m_motorOutputs/m_opMode <-> RxPdoMappingCspCsv/Modes of operation
//     TaskSlaveArmControl Outputs/SlaveArmControl.m_slaveRobot.m_slaveArms[3].m_joints[8].m_motorOutputs/m_cmdCurrent <-> RxPdoMappingCspCsv/Target Torque value
//     TaskSlaveArmControl Outputs/SlaveArmControl.m_slaveRobot.m_slaveArms[3].m_joints[8].m_motorOutputs/m_cmdMotorEncoder <-> RxPdoMappingCspCsv/Target position
//   SlaveController/SlaveController Instance <-> SlaveArm4/SetupJoint12
//     TaskSetupArmControl Inputs/SetupArmControl.m_setupRobot.m_setupArms[4].m_joints[1].m_motorInputs/m_linkEncoder <-> TxPdoMappingCspCsv/ENC2
//     TaskSetupArmControl Inputs/SetupArmControl.m_setupRobot.m_setupArms[4].m_joints[1].m_motorInputs/m_statusWord <-> TxPdoMappingCspCsv/Statusword
//     TaskSetupArmControl Inputs/SetupArmControl.m_setupRobot.m_setupArms[4].m_joints[2].m_motorInputs/m_statusWord <-> TxPdoMappingCspCsv/Statusword
//     TaskSetupArmControl Inputs/SetupArmControl.m_setupRobot.m_setupArms[4].m_joints[2].m_motorInputs/m_linkEncoder <-> TxPdoMappingCspCsv/Torque actual value
//     TaskSetupArmControl Outputs/SetupArmControl.m_setupRobot.m_setupArms[4].m_joints[1].m_motorOutputs/m_controlWord <-> RxPdoMappingCspCsv/Controlword
//   SlaveController/SlaveController Instance <-> SlaveArm4/SetupJoint3
//     TaskSetupArmControl Inputs/SetupArmControl.m_setupRobot.m_setupArms[4].m_joints[3].m_motorInputs/m_current <-> TxPdoMappingCspCsv/Torque actual value
//     TaskSetupArmControl Inputs/SetupArmControl.m_setupRobot.m_setupArms[4].m_joints[3].m_motorInputs/m_linkEncoder <-> TxPdoMappingCspCsv/ENC2
//     TaskSetupArmControl Inputs/SetupArmControl.m_setupRobot.m_setupArms[4].m_joints[3].m_motorInputs/m_motorEncoder <-> TxPdoMappingCspCsv/Position actual value
//     TaskSetupArmControl Inputs/SetupArmControl.m_setupRobot.m_setupArms[4].m_joints[3].m_motorInputs/m_statusWord <-> TxPdoMappingCspCsv/Statusword
//     TaskSetupArmControl Outputs/SetupArmControl.m_setupRobot.m_setupArms[4].m_joints[3].m_motorOutputs/m_cmdCurrent <-> RxPdoMappingCspCsv/Target torque
//     TaskSetupArmControl Outputs/SetupArmControl.m_setupRobot.m_setupArms[4].m_joints[3].m_motorOutputs/m_cmdMotorEncoder <-> RxPdoMappingCspCsv/Target position
//     TaskSetupArmControl Outputs/SetupArmControl.m_setupRobot.m_setupArms[4].m_joints[3].m_motorOutputs/m_controlWord <-> RxPdoMappingCspCsv/Controlword
//     TaskSetupArmControl Outputs/SetupArmControl.m_setupRobot.m_setupArms[4].m_joints[3].m_motorOutputs/m_opMode <-> RxPdoMappingCspCsv/Modes of operation
//   SlaveController/SlaveController Instance <-> SlaveArm4/SetupJoint4
//     TaskSetupArmControl Inputs/SetupArmControl.m_setupRobot.m_setupArms[4].m_joints[4].m_motorInputs/m_current <-> TxPdoMappingCspCsv/Torque actual value
//     TaskSetupArmControl Inputs/SetupArmControl.m_setupRobot.m_setupArms[4].m_joints[4].m_motorInputs/m_motorEncoder <-> TxPdoMappingCspCsv/Position actual value
//     TaskSetupArmControl Inputs/SetupArmControl.m_setupRobot.m_setupArms[4].m_joints[4].m_motorInputs/m_statusWord <-> TxPdoMappingCspCsv/Statusword
//     TaskSetupArmControl Outputs/SetupArmControl.m_setupRobot.m_setupArms[4].m_joints[4].m_motorOutputs/m_cmdCurrent <-> RxPdoMappingCspCsv/Target torque
//     TaskSetupArmControl Outputs/SetupArmControl.m_setupRobot.m_setupArms[4].m_joints[4].m_motorOutputs/m_cmdMotorEncoder <-> RxPdoMappingCspCsv/Target position
//     TaskSetupArmControl Outputs/SetupArmControl.m_setupRobot.m_setupArms[4].m_joints[4].m_motorOutputs/m_controlWord <-> RxPdoMappingCspCsv/Controlword
//     TaskSetupArmControl Outputs/SetupArmControl.m_setupRobot.m_setupArms[4].m_joints[4].m_motorOutputs/m_opMode <-> RxPdoMappingCspCsv/Modes of operation
//   SlaveController/SlaveController Instance <-> SlaveArm4/SetupJoint5
//     TaskSetupArmControl Inputs/SetupArmControl.m_setupRobot.m_setupArms[4].m_joints[4].m_motorInputs/m_linkEncoder <-> TxPdoMappingCspCsv/ENC2
//     TaskSetupArmControl Inputs/SetupArmControl.m_setupRobot.m_setupArms[4].m_joints[5].m_motorInputs/m_current <-> TxPdoMappingCspCsv/Torque actual value
//     TaskSetupArmControl Inputs/SetupArmControl.m_setupRobot.m_setupArms[4].m_joints[5].m_motorInputs/m_linkEncoder <-> TxPdoMappingCspCsv/analog input
//     TaskSetupArmControl Inputs/SetupArmControl.m_setupRobot.m_setupArms[4].m_joints[5].m_motorInputs/m_motorEncoder <-> TxPdoMappingCspCsv/Position actual value
//     TaskSetupArmControl Inputs/SetupArmControl.m_setupRobot.m_setupArms[4].m_joints[5].m_motorInputs/m_statusWord <-> TxPdoMappingCspCsv/Statusword
//     TaskSetupArmControl Outputs/SetupArmControl.m_setupRobot.m_setupArms[4].m_joints[5].m_motorOutputs/m_cmdCurrent <-> RxPdoMappingCspCsv/Target torque
//     TaskSetupArmControl Outputs/SetupArmControl.m_setupRobot.m_setupArms[4].m_joints[5].m_motorOutputs/m_cmdMotorEncoder <-> RxPdoMappingCspCsv/Target position
//     TaskSetupArmControl Outputs/SetupArmControl.m_setupRobot.m_setupArms[4].m_joints[5].m_motorOutputs/m_controlWord <-> RxPdoMappingCspCsv/Controlword
//     TaskSetupArmControl Outputs/SetupArmControl.m_setupRobot.m_setupArms[4].m_joints[5].m_motorOutputs/m_opMode <-> RxPdoMappingCspCsv/Modes of operation
//   SlaveController/SlaveController Instance <-> SlaveArm4/SlaveJoint1
//     TaskSlaveArmControl Inputs/SlaveArmControl.m_slaveRobot.m_slaveArms[4].m_joints[1].m_motorInputs/m_current <-> TxPdoMappingCspCsv/Torque actual value
//     TaskSlaveArmControl Inputs/SlaveArmControl.m_slaveRobot.m_slaveArms[4].m_joints[1].m_motorInputs/m_linkEncoder <-> TxPdoMappingCspCsv/ENC2
//     TaskSlaveArmControl Inputs/SlaveArmControl.m_slaveRobot.m_slaveArms[4].m_joints[1].m_motorInputs/m_motorEncoder <-> TxPdoMappingCspCsv/Position actual value
//     TaskSlaveArmControl Inputs/SlaveArmControl.m_slaveRobot.m_slaveArms[4].m_joints[1].m_motorInputs/m_statusWord <-> TxPdoMappingCspCsv/Statusword
//     TaskSlaveArmControl Outputs/SlaveArmControl.m_slaveRobot.m_slaveArms[4].m_joints[1].m_motorOutputs/m_cmdCurrent <-> RxPdoMappingCspCsv/Target torque
//     TaskSlaveArmControl Outputs/SlaveArmControl.m_slaveRobot.m_slaveArms[4].m_joints[1].m_motorOutputs/m_cmdMotorEncoder <-> RxPdoMappingCspCsv/Target position
//     TaskSlaveArmControl Outputs/SlaveArmControl.m_slaveRobot.m_slaveArms[4].m_joints[1].m_motorOutputs/m_controlWord <-> RxPdoMappingCspCsv/Controlword
//     TaskSlaveArmControl Outputs/SlaveArmControl.m_slaveRobot.m_slaveArms[4].m_joints[1].m_motorOutputs/m_opMode <-> RxPdoMappingCspCsv/Modes of operation
//   SlaveController/SlaveController Instance <-> SlaveArm4/SlaveJoint2
//     TaskCartControl Inputs/CartControl.m_cartRobot.m_slaveCart.m_carRotaOverhangIO[4] <-> TxPdoMappingCspCsv/digital input
//     TaskSetupArmControl Outputs/SetupArmControl.m_setupRobot.m_setupArms[4].m_lightIO <-> RxPdoMappingCspCsv/Target velocity
//     TaskSlaveArmControl Inputs/SlaveArmControl.m_slaveRobot.m_slaveArms[4].m_joints[2].m_motorInputs/m_current <-> TxPdoMappingCspCsv/Torque actual value
//     TaskSlaveArmControl Inputs/SlaveArmControl.m_slaveRobot.m_slaveArms[4].m_joints[2].m_motorInputs/m_linkEncoder <-> TxPdoMappingCspCsv/ENC2
//     TaskSlaveArmControl Inputs/SlaveArmControl.m_slaveRobot.m_slaveArms[4].m_joints[2].m_motorInputs/m_motorEncoder <-> TxPdoMappingCspCsv/Position actual value
//     TaskSlaveArmControl Inputs/SlaveArmControl.m_slaveRobot.m_slaveArms[4].m_joints[2].m_motorInputs/m_statusWord <-> TxPdoMappingCspCsv/Statusword
//     TaskSlaveArmControl Outputs/SlaveArmControl.m_slaveRobot.m_slaveArms[4].m_joints[2].m_motorOutputs/m_cmdCurrent <-> RxPdoMappingCspCsv/Target torque
//     TaskSlaveArmControl Outputs/SlaveArmControl.m_slaveRobot.m_slaveArms[4].m_joints[2].m_motorOutputs/m_cmdMotorEncoder <-> RxPdoMappingCspCsv/Target position
//     TaskSlaveArmControl Outputs/SlaveArmControl.m_slaveRobot.m_slaveArms[4].m_joints[2].m_motorOutputs/m_controlWord <-> RxPdoMappingCspCsv/Controlword
//     TaskSlaveArmControl Outputs/SlaveArmControl.m_slaveRobot.m_slaveArms[4].m_joints[2].m_motorOutputs/m_opMode <-> RxPdoMappingCspCsv/Modes of operation
//   SlaveController/SlaveController Instance <-> SlaveArm4/SlaveJoint3
//     TaskCartControl Inputs/CartControl.m_cartRobot.m_slaveCart.m_trocarIO[4] <-> TxPdoMappingCspCsv/digital input
//     TaskSetupArmControl Inputs/SetupArmControl.m_setupRobot.m_setupArms[4].m_adjustIO <-> TxPdoMappingCspCsv/digital input
//     TaskSlaveArmControl Inputs/SlaveArmControl.m_slaveRobot.m_slaveArms[4].m_adjustIO <-> TxPdoMappingCspCsv/digital input
//     TaskSlaveArmControl Inputs/SlaveArmControl.m_slaveRobot.m_slaveArms[4].m_joints[3].m_motorInputs/m_current <-> TxPdoMappingCspCsv/Torque actual value
//     TaskSlaveArmControl Inputs/SlaveArmControl.m_slaveRobot.m_slaveArms[4].m_joints[3].m_motorInputs/m_linkEncoder <-> TxPdoMappingCspCsv/ENC2 for aix1
//     TaskSlaveArmControl Inputs/SlaveArmControl.m_slaveRobot.m_slaveArms[4].m_joints[3].m_motorInputs/m_motorEncoder <-> TxPdoMappingCspCsv/Position actual value
//     TaskSlaveArmControl Inputs/SlaveArmControl.m_slaveRobot.m_slaveArms[4].m_joints[3].m_motorInputs/m_statusWord <-> TxPdoMappingCspCsv/Statusword
//     TaskSlaveArmControl Outputs/SlaveArmControl.m_slaveRobot.m_slaveArms[4].m_joints[3].m_motorOutputs/m_cmdCurrent <-> RxPdoMappingCspCsv/Target Torque value
//     TaskSlaveArmControl Outputs/SlaveArmControl.m_slaveRobot.m_slaveArms[4].m_joints[3].m_motorOutputs/m_cmdMotorEncoder <-> RxPdoMappingCspCsv/Target position
//     TaskSlaveArmControl Outputs/SlaveArmControl.m_slaveRobot.m_slaveArms[4].m_joints[3].m_motorOutputs/m_controlWord <-> RxPdoMappingCspCsv/Controlword
//     TaskSlaveArmControl Outputs/SlaveArmControl.m_slaveRobot.m_slaveArms[4].m_joints[3].m_motorOutputs/m_opMode <-> RxPdoMappingCspCsv/Modes of operation
//   SlaveController/SlaveController Instance <-> SlaveArm4/SlaveJoint45
//     TaskSlaveArmControl Inputs/SlaveArmControl.m_slaveRobot.m_slaveArms[4].m_joints[4].m_motorInputs/m_current <-> TxPdoMappingCspCsv/Velocity actual value for aix2
//     TaskSlaveArmControl Inputs/SlaveArmControl.m_slaveRobot.m_slaveArms[4].m_joints[5].m_motorInputs/m_current <-> TxPdoMappingCspCsv/Velocity actual value for aix3
//     TaskSlaveArmControl Inputs/SlaveArmControl.m_slaveRobot.m_slaveArms[4].m_joints[4].m_motorInputs/m_linkEncoder <-> TxPdoMappingCspCsv/ENC2 for aix2
//     TaskSlaveArmControl Inputs/SlaveArmControl.m_slaveRobot.m_slaveArms[4].m_joints[5].m_motorInputs/m_linkEncoder <-> TxPdoMappingCspCsv/ENC2 for aix3
//     TaskSlaveArmControl Inputs/SlaveArmControl.m_slaveRobot.m_slaveArms[4].m_joints[4].m_motorInputs/m_motorEncoder <-> TxPdoMappingCspCsv/Position actual value for aix2
//     TaskSlaveArmControl Inputs/SlaveArmControl.m_slaveRobot.m_slaveArms[4].m_joints[5].m_motorInputs/m_motorEncoder <-> TxPdoMappingCspCsv/Position actual value for aix3
//     TaskSlaveArmControl Inputs/SlaveArmControl.m_slaveRobot.m_slaveArms[4].m_joints[4].m_motorInputs/m_statusWord <-> TxPdoMappingCspCsv/Statusword
//     TaskSlaveArmControl Inputs/SlaveArmControl.m_slaveRobot.m_slaveArms[4].m_joints[5].m_motorInputs/m_statusWord <-> TxPdoMappingCspCsv/Statusword
//     TaskSlaveArmControl Inputs/SlaveArmControl.m_slaveRobot.m_slaveArms[4].m_panelInstrumentOnIO <-> TxPdoMappingCspCsv/digital input
//     TaskSlaveArmControl Outputs/SlaveArmControl.m_slaveRobot.m_slaveArms[4].m_joints[4].m_motorOutputs/m_cmdCurrent <-> RxPdoMappingCspCsv/Target Torque value for aix2
//     TaskSlaveArmControl Outputs/SlaveArmControl.m_slaveRobot.m_slaveArms[4].m_joints[5].m_motorOutputs/m_cmdCurrent <-> RxPdoMappingCspCsv/Target Torque value for aix3
//     TaskSlaveArmControl Outputs/SlaveArmControl.m_slaveRobot.m_slaveArms[4].m_joints[4].m_motorOutputs/m_cmdMotorEncoder <-> RxPdoMappingCspCsv/Target position value for aix2
//     TaskSlaveArmControl Outputs/SlaveArmControl.m_slaveRobot.m_slaveArms[4].m_joints[5].m_motorOutputs/m_cmdMotorEncoder <-> RxPdoMappingCspCsv/Target position value for aix3
//     TaskSlaveArmControl Outputs/SlaveArmControl.m_slaveRobot.m_slaveArms[4].m_joints[4].m_motorOutputs/m_controlWord <-> RxPdoMappingCspCsv/Controlword
//     TaskSlaveArmControl Outputs/SlaveArmControl.m_slaveRobot.m_slaveArms[4].m_joints[4].m_motorOutputs/m_opMode <-> RxPdoMappingCspCsv/Modes of operation
//   SlaveController/SlaveController Instance <-> SlaveArm4/SlaveJoint678
//     TaskSlaveArmControl Inputs/SlaveArmControl.m_slaveRobot.m_slaveArms[4].m_joints[6].m_motorInputs/m_current <-> TxPdoMappingCspCsv/Velocity actual value for aix2
//     TaskSlaveArmControl Inputs/SlaveArmControl.m_slaveRobot.m_slaveArms[4].m_joints[7].m_motorInputs/m_current <-> TxPdoMappingCspCsv/Velocity actual value for aix3
//     TaskSlaveArmControl Inputs/SlaveArmControl.m_slaveRobot.m_slaveArms[4].m_joints[6].m_motorInputs/m_linkEncoder <-> TxPdoMappingCspCsv/ENC2 for aix2
//     TaskSlaveArmControl Inputs/SlaveArmControl.m_slaveRobot.m_slaveArms[4].m_joints[7].m_motorInputs/m_linkEncoder <-> TxPdoMappingCspCsv/ENC2 for aix3
//     TaskSlaveArmControl Inputs/SlaveArmControl.m_slaveRobot.m_slaveArms[4].m_joints[8].m_motorInputs/m_linkEncoder <-> TxPdoMappingCspCsv/ENC2 for aix1
//     TaskSlaveArmControl Inputs/SlaveArmControl.m_slaveRobot.m_slaveArms[4].m_joints[6].m_motorInputs/m_motorEncoder <-> TxPdoMappingCspCsv/Position actual value for aix2
//     TaskSlaveArmControl Inputs/SlaveArmControl.m_slaveRobot.m_slaveArms[4].m_joints[7].m_motorInputs/m_motorEncoder <-> TxPdoMappingCspCsv/Position actual value for aix3
//     TaskSlaveArmControl Inputs/SlaveArmControl.m_slaveRobot.m_slaveArms[4].m_joints[6].m_motorInputs/m_statusWord <-> TxPdoMappingCspCsv/Statusword
//     TaskSlaveArmControl Inputs/SlaveArmControl.m_slaveRobot.m_slaveArms[4].m_joints[7].m_motorInputs/m_statusWord <-> TxPdoMappingCspCsv/Statusword
//     TaskSlaveArmControl Inputs/SlaveArmControl.m_slaveRobot.m_slaveArms[4].m_joints[8].m_motorInputs/m_statusWord <-> TxPdoMappingCspCsv/Statusword
//     TaskSlaveArmControl Inputs/SlaveArmControl.m_slaveRobot.m_slaveArms[4].m_joints[8].m_motorInputs/m_current <-> TxPdoMappingCspCsv/Torque actual value
//     TaskSlaveArmControl Inputs/SlaveArmControl.m_slaveRobot.m_slaveArms[4].m_joints[8].m_motorInputs/m_motorEncoder <-> TxPdoMappingCspCsv/Position actual value
//     TaskSlaveArmControl Outputs/SlaveArmControl.m_slaveRobot.m_slaveArms[4].m_joints[6].m_motorOutputs/m_cmdCurrent <-> RxPdoMappingCspCsv/Target Torque value for aix2
//     TaskSlaveArmControl Outputs/SlaveArmControl.m_slaveRobot.m_slaveArms[4].m_joints[7].m_motorOutputs/m_cmdCurrent <-> RxPdoMappingCspCsv/Target Torque value for aix3
//     TaskSlaveArmControl Outputs/SlaveArmControl.m_slaveRobot.m_slaveArms[4].m_joints[6].m_motorOutputs/m_cmdMotorEncoder <-> RxPdoMappingCspCsv/Target position value for aix2
//     TaskSlaveArmControl Outputs/SlaveArmControl.m_slaveRobot.m_slaveArms[4].m_joints[7].m_motorOutputs/m_cmdMotorEncoder <-> RxPdoMappingCspCsv/Target position value for aix3
//     TaskSlaveArmControl Outputs/SlaveArmControl.m_slaveRobot.m_slaveArms[4].m_joints[6].m_motorOutputs/m_controlWord <-> RxPdoMappingCspCsv/Controlword
//     TaskSlaveArmControl Outputs/SlaveArmControl.m_slaveRobot.m_slaveArms[4].m_joints[6].m_motorOutputs/m_opMode <-> RxPdoMappingCspCsv/Modes of operation
//     TaskSlaveArmControl Outputs/SlaveArmControl.m_slaveRobot.m_slaveArms[4].m_joints[8].m_motorOutputs/m_cmdCurrent <-> RxPdoMappingCspCsv/Target Torque value
//     TaskSlaveArmControl Outputs/SlaveArmControl.m_slaveRobot.m_slaveArms[4].m_joints[8].m_motorOutputs/m_cmdMotorEncoder <-> RxPdoMappingCspCsv/Target position
//   SlaveController/SlaveController Instance <-> SlaveController/SlaveController Instance
//     TaskCartControl Inputs/CartControl.m_cartDataPool.m_safetyData <-> TaskCartControl Outputs/SafetyCheck.m_safetyCheckData
//     TaskCartControl Inputs/CartControl.m_cartDataPool.m_slaveStatus <-> TaskSlaveArmControl Outputs/SlaveArmControl.m_slaveStatus
//     TaskDynamic Inputs/RobotDynamics.m_instruInfo <-> TaskSlaveArmControl Outputs/SlaveArmControl.m_slaveStatus/m_instruStauts
//     TaskDynamic Inputs/RobotDynamics.m_setupJointData <-> TaskSetupArmControl Outputs/SetupArmControl.m_setupJointsData
//     TaskDynamic Inputs/RobotDynamics.m_slaveJointsData <-> TaskSlaveArmControl Outputs/SlaveArmControl.m_slaveJointsData
//     TaskSafetyCheck Inputs/SafetyCheck.m_cartJointsData <-> TaskCartControl Outputs/CartControl.m_cartJointsData
//     TaskSafetyCheck Inputs/SafetyCheck.m_cartStatus <-> TaskCartControl Outputs/CartControl.m_cartStatus
//     TaskSafetyCheck Inputs/SafetyCheck.m_setupJointsData <-> TaskSetupArmControl Outputs/SetupArmControl.m_setupJointsData
//     TaskSafetyCheck Inputs/SafetyCheck.m_setupStatus <-> TaskSlaveArmControl Outputs/SetupArmControl.m_setupStatus
//     TaskSafetyCheck Inputs/SafetyCheck.m_slaveJointData <-> TaskSlaveArmControl Outputs/SlaveArmControl.m_slaveJointsData
//     TaskSafetyCheck Inputs/SafetyCheck.m_slaveStatus <-> TaskSlaveArmControl Outputs/SlaveArmControl.m_slaveStatus
//     TaskSetupArmControl Inputs/SetupArmControl.m_setupInputDataPool.m_safetyData <-> TaskCartControl Outputs/SafetyCheck.m_safetyCheckData
//     TaskSetupArmControl Inputs/SetupArmControl.m_setupInputDataPool.m_setupJnt3Gravity <-> TaskDynamic Outputs/RobotDynamics.m_setupJnt3Gravity
//     TaskSetupArmControl Inputs/SetupArmControl.m_setupInputDataPool.m_setupJnt5Gravity <-> TaskDynamic Outputs/RobotDynamics.m_setupJnt5Gravity
//     TaskSetupArmControl Inputs/SetupArmControl.m_setupInputDataPool.m_slaveStatus <-> TaskSlaveArmControl Outputs/SlaveArmControl.m_slaveStatus
//     TaskSlaveArmControl Inputs/SlaveArmControl.m_slaveInputDataPool.m_safetyData <-> TaskCartControl Outputs/SafetyCheck.m_safetyCheckData
//     TaskSlaveArmControl Inputs/SlaveArmControl.m_slaveInputDataPool.m_setupStatus <-> TaskSlaveArmControl Outputs/SetupArmControl.m_setupStatus
//     TaskSlaveArmControl Inputs/SlaveArmControl.m_slaveInputDataPool.m_slaveDynaData <-> TaskDynamic Outputs/RobotDynamics.m_slaveDynaData

CONFIGURATION SlaveController
    RESOURCE PLC ON TwinCAT3
        TASK TaskCartControl(INTERVAL := T#1ms, PRIORITY := 4);
        TASK TaskSafetyCheck(INTERVAL := T#1ms, PRIORITY := 6);
        TASK TaskSlaveArmControl(INTERVAL := T#250us, PRIORITY := 1);
        PROGRAM CartControl WITH TaskCartControl : CartControl;
        PROGRAM SafetyCheck WITH TaskSafetyCheck : SafetyCheck;
        PROGRAM SlaveArmControl WITH TaskSlaveArmControl : SlaveArmControl;
    END_RESOURCE
END_CONFIGURATION

// ---- DUTs/Enum/E_ArmLightCtrlWord.TcDUT
//*******************机械臂与动力盒上的灯光写入********************
//不可恢复性故障-----红色常亮
//可恢复故障----琥珀色-先闪烁5s、再进行常亮
//正处于器械控制或者端口控制状态-----蓝色闪烁
//该手术臂正在执行一项需要用户短时间等待的活动、例如器械卡接----蓝色-脉动闪烁
//工具更换引导正在进行中-----绿色闪烁
//未通电、已禁用、已收起----------关
//系统正常运行-----蓝色常亮
//灯光颜色--0-灯灭、1蓝灯常亮、2蓝灯闪烁、3琥珀色闪烁、4红灯闪烁、5绿灯常亮、6绿灯闪烁、7红灯常亮、8琥珀色常亮、9蓝灯脉动式闪烁
TYPE E_ArmLightCtrlWord :
(
	ArmLight_Off := 0,
	ArmLight_BlueOn :=1,
	ArmLight_BlueBlink :=2,
	ArmLight_AmberBlink :=3,
	ArmLight_RedBlink :=4,
	ArmLight_GreenOn :=5,
	ArmLight_GreenBlink :=6,
	ArmLight_redOn :=7,
	ArmLight_AmberOn :=8,
	ArmLight_BluePulse :=9
);
END_TYPE

// ---- DUTs/Enum/E_CartJointState.TcDUT
TYPE E_CartJointState :
(
	CartJointState_Error := 1,
	CartJointState_Init := 2,
	CartJointState_SelfCheck := 3,
	CartJointState_Standby := 4,
	CartJointState_Ready := 5,
	CartJointState_InSurgery := 6,
	CartJointState_SteadyFootDeployment := 7,
	CartJointState_Movement := 8,
	CartJointState_HangAdjust := 9,
	CartJointState_AsepticDeployment := 10,
	CartJointState_RotaOverhang := 11,
	CartJointState_SlowStop := 12,
	CartJointState_StandColuAdjust := 13,
	
	CartJointState_totalNum := CartJointState_StandColuAdjust
);
END_TYPE

// ---- DUTs/Enum/E_EndoscopeType.TcDUT
TYPE E_EndoscopeType :
(
	EndoscopeType_0:=1,
	EndoScopeType_30:=2
);
END_TYPE

// ---- DUTs/Enum/E_EndoscopePosture.TcDUT
TYPE E_EndoscopePosture:
(
	EndoscopePosture_HeadUp:=1,
	EndoScopePosture_HeadDown:=2
);
END_TYPE

// ---- DUTs/Enum/E_InstrumentType.TcDUT
TYPE E_InstrumentType :
(
	InstruType_UNKNOWM := 0,
	InstruType_CadiereForceps :=7,
	InstruType_NeedleDriver :=8,
	InstruType_MegaSCNeedleDriver :=9,// mega suture-cut needle driver
	InstruType_SCNeedleDriver :=10, // suture-cut needle driver
	InstruType_RoundTipScissors :=11,
	InstruType_ProGraspForceps :=12,
	InstruType_MarylandForceps :=13, // Maryland bipolar forceps
	InstruType_FenestratedForceps :=14, // Fnestrated bipolar forceps
	InstruType_CurvedScissors :=15, // monopolar curved scissors
	InstruType_CauteryHook :=16,
	InstruType_CauterySpatula :=17,
	InstruType_Endoscope := 20,
	InstruType_NewEndoscope := 31,
	InstruType_UltrasoundKnifeS :=42,
	InstruType_UltrasoundKnifeU :=43,
	InstruType_TipUpFenestratedGrasper :=44,
	InstruType_MegaNeedleDriver :=45,
	InstruType_DeBakeyForceps :=46,
	InstruType_BlackDiamondForceps :=47,
	InstruType_PottsScissors :=48,
	InstruType_CurvedBipolarDissector :=49,
	InstruType_MicroBipolarForceps :=50,
	InstruType_ForceBipolar :=51,
	InstruType_MicroCauteryHook :=52
);
END_TYPE

// ---- DUTs/Enum/E_MasterArmState.TcDUT
// Notice: Each state has a corresponding controller, which has a fixed index.
// Add the new state at the end and update the total num
TYPE E_MasterArmState :
(
	MasterArmState_Error := 1,
	MasterArmState_Init :=2,
	MasterArmState_Home :=3,
	MasterArmState_Standby :=4,
	MasterArmState_Matching :=5,
	MasterArmState_Ready :=6,
	MasterArmState_MasterSlave :=7,
	MasterArmState_Clutch :=8,
	MasterArmState_Endoscope :=9,
	MasterArmState_Cart := 10,
	MasterArmState_GravityCali := 11,
	MasterArmState_Test :=12,
	
	MasterArmState_totalNum :=MasterArmState_Test

);
END_TYPE

// ---- DUTs/Enum/E_SetupArmState.TcDUT
TYPE E_SetupArmState :
(
	SetupArmState_Error := 1,
	SetupArmState_Init :=2,
	SetupArmState_SelfCheck :=3,
	SetupArmState_Hold :=4,
	SetupArmState_ManualAdjust :=5,
	SetupArmState_AutoAdjust :=6,
	SetupArmState_Package :=7,
	SetupArmState_Cart := 8,
	SetupArmState_jnt3GravityCali := 9,
	SetupArmState_jnt5GravityCali := 10,
	SetupArmState_Disable := 11,
	SetupArmState_Performance:=12,
	
	SetupArmState_totalNum :=SetupArmState_Performance
);
END_TYPE

// ---- DUTs/Enum/E_SlaveArmState.TcDUT
TYPE E_SlaveArmState :
(
	SlaveArmState_Error := 1,
	SlaveArmState_Init :=2,
	SlaveArmState_SelfCheck :=3,
	SlaveArmState_Standby :=4,
	SlaveArmState_MountPanel:=5,
	SlaveArmState_PanelReady :=6,
	SlaveArmState_MountInstru :=7,
	SlaveArmState_InstruReady :=8,
	SlaveArmState_MasterSlave :=9,
	SlaveArmState_ScopeReady :=10,
	SlaveArmState_EndoScope :=11,
	SlaveArmState_Adjust :=12,
	SlaveArmState_Package :=13,
	SlaveArmState_Cart := 14,
	SlaveArmState_GravityCali := 15,
	SlaveArmState_Test := 16,
	SlaveArmState_InstruRetract :=17,
	SlaveArmState_InstruInvasion :=18,
	SlaveArmState_Disable := 19,
	SlaveArmState_InstruCali := 20,
	SlaveArmState_ScopeToggle :=21,
	SlaveArmState_Performance:=22,
	SlaveArmState_Stop :=23,
	
	SlaveArmState_totalNum :=SlaveArmState_Stop
);
END_TYPE

// ---- DUTs/Structure/MasterSlaveCommunication/ST_MasterStatus.TcDUT
// Input from master arm control task, including arm status and cartesian data
TYPE ST_MasterStatus :
STRUCT
	// master heart beat
	m_masterHeartBeat :INT:=0;
	
	// self-check trigger flag
	m_slaveSelfCheckFlag :BOOL :=FALSE;
	
	// linear motion scale
	m_motionScale : LREAL:=1.5;
	
	// state machine
	m_armState:ARRAY[1..g_mArmNum] OF E_masterArmState;
	
	// index(0 to 4) of slave arm which is tele-linked to master arm
	m_teleSlaveArmIdx :ARRAY[1..g_mArmNum] OF E_MatchedSlaveArmIdx;
	
	// grip angle
	m_gripAngle:ARRAY[1..g_mArmNum] OF LREAL;
	
	// current arm pose in monitor coordinate
	m_curArmPose:ARRAY[1..g_mArmNum] OF ST_Frame;
	
	// current arm twist[linear velocity; angular veloicty] in monitor coordinate
	m_curArmTwist:ARRAY[1..g_mArmNum] OF Vec6d;
	
	//master pedal hover 
	m_pedalHover : ARRAY [1..2] OF BOOL;
	
	// electric Knife Pedal Trigger 
	m_electricKnifePedalTrigger : ARRAY [1..2] OF UINT;
	
	//Attempt to enter master-slave control 
	m_tryMSControl : ARRAY [1..2] OF INT;
	
	//master robot stop button trigger flag
	m_masterStopButton : BOOL;
	
	// ui send fault reset flag from master
	m_uiResetFault : UINT;
END_STRUCT
END_TYPE

// ---- DUTs/Structure/MasterSlaveCommunication/ST_SlaveStatus.TcDUT
// Output from slave arm control task, including arm status and cartesian data
// Input to safety task and Master controller
TYPE ST_SlaveStatus :
STRUCT
	
	// state machine
	m_armState:ARRAY[1..g_sArmNum] OF E_SlaveArmState:=[g_sArmNum(SlaveArmState_Error)];
	
	// self-check pass flag
	m_selfCheckPass :ARRAY[1..g_sArmNum] OF BOOL :=[4(False)];
	
	// instrument info
	m_instruStauts :ARRAY[1..g_sArmNum] OF ST_InstruStatus;
	
	// flag if endoscope is mounted
	m_endoscopeMounted :BOOL := FALSE;
	
	// endoscope pose in cart coordinate
	m_endoscopePose : ST_Frame;
	
	// command arm pose in slave arm coordinate
	m_cmdArmPose:ARRAY[1..g_sArmNum] OF ST_Frame;
	
	// current arm pose in slave arm coordinate
	m_curArmPose:ARRAY[1..g_sArmNum] OF ST_Frame;
	
	// simulation arm pose in slave arm coordinate
	m_simArmPose:ARRAY[1..g_sArmNum] OF ST_Frame;
	
	// master slave pose error [position, angle*axis] in endoscope coordinate
	m_masterSlavePoseError :ARRAY[1..g_sArmNum] OF Vec6d; 

	//read instrument information error ID
	m_instruReadErrId : ARRAY[1..g_sArmNum] OF INT;
	
	//instrument install status
	m_instruInstallStatus : ARRAY[1..g_sArmNum] OF BOOL;
	
	//instrument clamp error Id 
	m_instruClampErrId : ARRAY[1..g_sArmNum] OF UINT;
	
	//panel install status
	m_panelInstallStatus : ARRAY[1..g_sArmNum] OF BOOL;
	
	//panel clamp error ID
	m_panelClampErrId : ARRAY[1..g_sArmNum] OF UINT;
	
	//trocar install status 
	m_trocarOnFlag : ARRAY[1..g_sArmNum] OF BOOL;

	// flag if master are connected
	m_masterOnLine :BOOL ;
	
	// slave robot stop button trigger 
	m_slaveStopButton : BOOL;
END_STRUCT
END_TYPE

// ---- DUTs/Structure/ST_CartInputDataPool.TcDUT
//TODO:  check if used
TYPE ST_CartInputDataPool :
STRUCT
	// safety information, import from safety check task
	m_safetyData AT %I*: ST_SafetyData;
	
	// slave status, import from slave control task
	m_slaveStatus AT %I*: ST_SlaveStatus;
	
	//UI information, import from UI controller
	m_UIData :ST_CartUIData;
	
	
END_STRUCT
END_TYPE

// ---- DUTs/Structure/ST_InstruOnChipData.TcDUT
TYPE ST_InstruOnChipData :
STRUCT

	// ID
	m_InstruID: INT:=0;
	
	// series number
	m_InstruseriesNum : ULINT:=0;
	
	// current and max usage counts
	m_InstruUsageCounts :ULINT;
	
	//Instrument Zero augular offset
	m_InstruPos:Vec5d;
	
	//Instrument state
	m_InstruReadSucceed:BOOL;
	
	//Instrument Clamp Error
	m_Error:BOOL;
	m_ErrorID:INT;//1器械类型错误、2器械使用次数超限、3两个内窥镜

END_STRUCT
END_TYPE

// ---- DUTs/Structure/ST_InstruTypeInfo.TcDUT
TYPE ST_InstruTypeInfo :
STRUCT
	//ID
	m_InstruID: INT:=0;
	
	// has one or two finger
	m_isSingleFinger:BOOL;
	
	// energy type
	m_energyType:UINT:=0;
	
	// name
	m_instruName : STRING:='null';
	m_instruNameCH : WSTRING:="无效器械";
	
	// max use number
	m_maxUseNum :UINT :=20;
	
	// instrument geometric parameters
	m_rodLength:LREAL:=0.5392;
	m_headLength:LREAL :=0.01;
	m_fingerLength:LREAL :=0;
	m_maxGripAngle :LREAL := 50.0 * g_deg2Rad;
	
	// instrument reduction parameters
	m_k1:LREAL:=1;
	m_k2:LREAL:=1;
	m_k3:LREAL:=1;
	
	// instrument wrist DH joint limit
	m_rollLimit:LREAL:=5.5;
	m_pitchLimit:LREAL:=75*g_deg2Rad;
	m_yawLimit:LREAL:=PI/2;
	
	// grip force (mA)
	m_normGripTrq :LREAL := 150;
	// instrument backlash
	m_instruYawBacklash :LREAL:=0.0;
	m_instruPitchBachlash :LREAL :=0.0;
END_STRUCT
END_TYPE

// ---- DUTs/Structure/ST_SetupInputDataPool.TcDUT
// Struct contains all data from other tasks and controller used for slave control
TYPE ST_SetupInputDataPool :
STRUCT
				
	// slave status, import from slave control task
	m_slaveStatus AT %I*: ST_SlaveStatus;
	
	// safety information, import from safety check task
	m_safetyData AT %I*: ST_SafetyData;
	
	// slave gravity
	m_setupJnt3Gravity AT %I* : ARRAY[1..g_sArmNum] OF LREAL;
	m_setupJnt5Gravity AT %I* :  ARRAY[1..g_sArmNum] of LREAL;
	
	
END_STRUCT
END_TYPE

// ---- DUTs/Structure/TasksCommunication/ST_CartJointData.TcDUT
TYPE ST_CartJointData :
STRUCT
	
	// joint position compute with motor encoder
	m_curMotorPos : Vec8d;
	
	// joint position compute with link/abs encoder
	m_curLinkPos : Vec8d;
	
	// target joint position 
	m_cmdJntPos : Vec8d;
	
	// current joint position 
	m_curJntPos : Vec8d;
	
	// target joint velocity 
	m_cmdJntVel : Vec8d;
	
	// current joint position 
	m_curJntVel : Vec8d;
	
	// command joint torque 
	m_cmdJntTrq : Vec8d;
	
	// current joint torque 
	m_curJntTrq : Vec8d;
	
END_STRUCT
END_TYPE

// ---- DUTs/Structure/TasksCommunication/ST_CartMotorInput.TcDUT
TYPE ST_CartMotorInput EXTENDS ST_MotorInputs :
STRUCT
	//
END_STRUCT
END_TYPE

// ---- DUTs/Structure/TasksCommunication/ST_CartMotorOutput.TcDUT
TYPE ST_CartMotorOutput  :
STRUCT
	//MingZhi drive ues
	m_cmdVelMz:DINT:=0;
	
	m_cmdAccMz:DINT:=0;
	
	m_cmdVelMzVelMode:DINT:=0;
	
	
END_STRUCT
END_TYPE

// ---- DUTs/Structure/TasksCommunication/ST_CartStatus.TcDUT
// Output from cart control task
// Input to slave arm control task  
TYPE ST_CartStatus :
STRUCT
	m_CartState :E_CartJointState:=CartJointState_Error;
	
	m_cartDumpEnergy :UINT;
	
